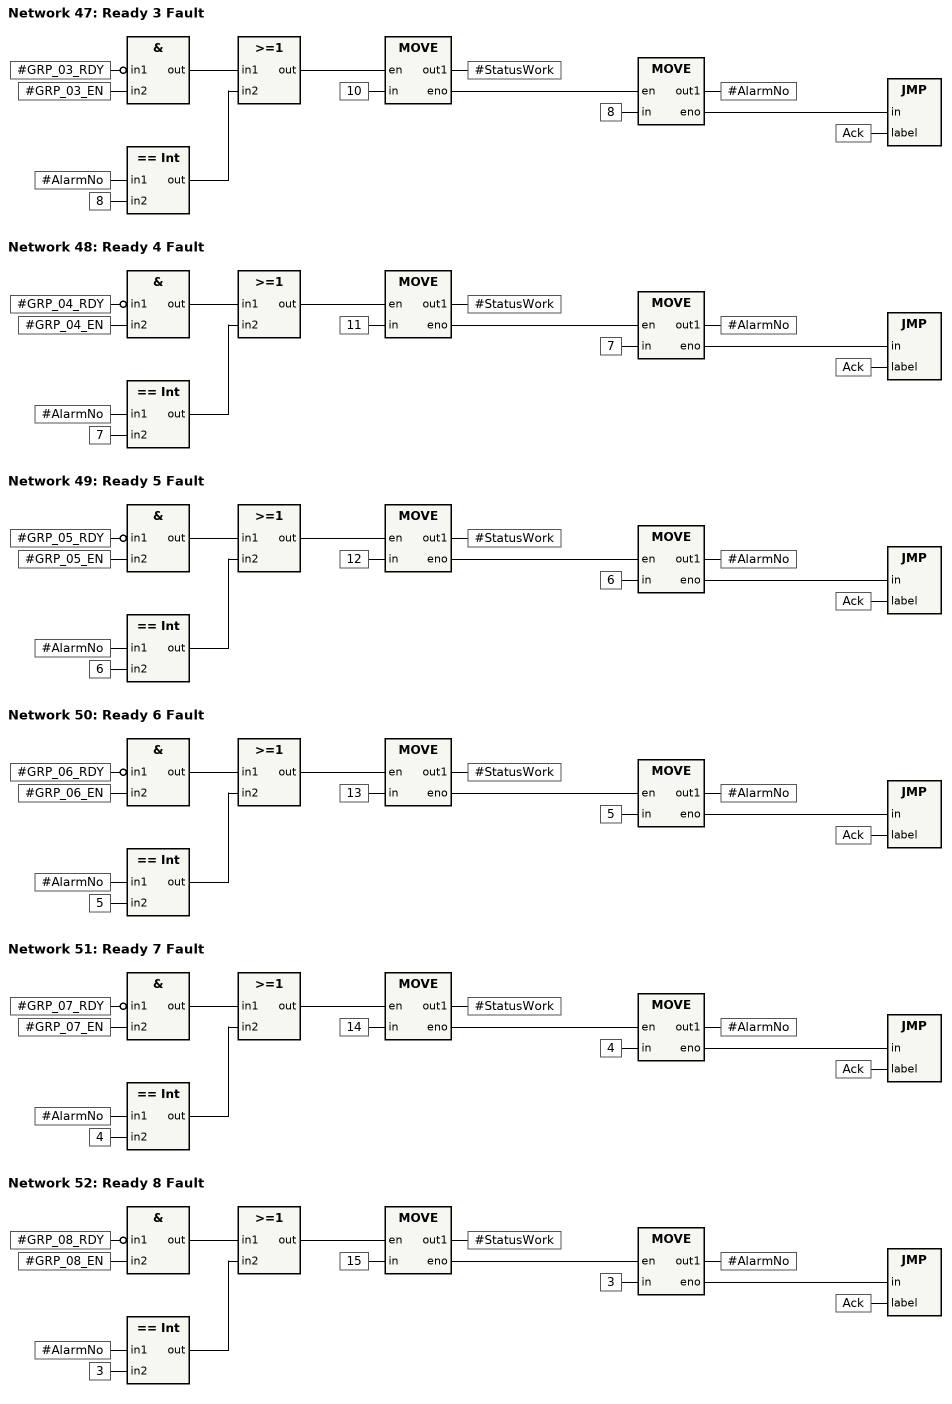
   // ENO of a box is taken as its EN; it also drops when the box reports an error
   #_w1 := (NOT #GRP_03_RDY AND #GRP_03_EN) OR (#AlarmNo = 8);
   IF #_w1 THEN
       #StatusWork := 10;
       #AlarmNo := 8;
       GOTO Ack;
   END_IF;
END_REGION

REGION Network 48: Ready 4 Fault
   // ENO of a box is taken as its EN; it also drops when the box reports an error
   #_w1 := (NOT #GRP_04_RDY AND #GRP_04_EN) OR (#AlarmNo = 7);
   IF #_w1 THEN
       #StatusWork := 11;
       #AlarmNo := 7;
       GOTO Ack;
   END_IF;
END_REGION

REGION Network 49: Ready 5 Fault
   // ENO of a box is taken as its EN; it also drops when the box reports an error
   #_w1 := (NOT #GRP_05_RDY AND #GRP_05_EN) OR (#AlarmNo = 6);
   IF #_w1 THEN
       #StatusWork := 12;
       #AlarmNo := 6;
       GOTO Ack;
   END_IF;
END_REGION

REGION Network 50: Ready 6 Fault
   // ENO of a box is taken as its EN; it also drops when the box reports an error
   #_w1 := (NOT #GRP_06_RDY AND #GRP_06_EN) OR (#AlarmNo = 5);
   IF #_w1 THEN
       #StatusWork := 13;
       #AlarmNo := 5;
       GOTO Ack;
   END_IF;
END_REGION

REGION Network 51: Ready 7 Fault
   // ENO of a box is taken as its EN; it also drops when the box reports an error
   #_w1 := (NOT #GRP_07_RDY AND #GRP_07_EN) OR (#AlarmNo = 4);
   IF #_w1 THEN
       #StatusWork := 14;
       #AlarmNo := 4;
       GOTO Ack;
   END_IF;
END_REGION

REGION Network 52: Ready 8 Fault
   // ENO of a box is taken as its EN; it also drops when the box reports an error
   #_w1 := (NOT #GRP_08_RDY AND #GRP_08_EN) OR (#AlarmNo = 3);
   IF #_w1 THEN
       #StatusWork := 15;
       #AlarmNo := 3;
       GOTO Ack;
   END_IF;
END_REGION

REGION Network 53: Ready 9 Fault
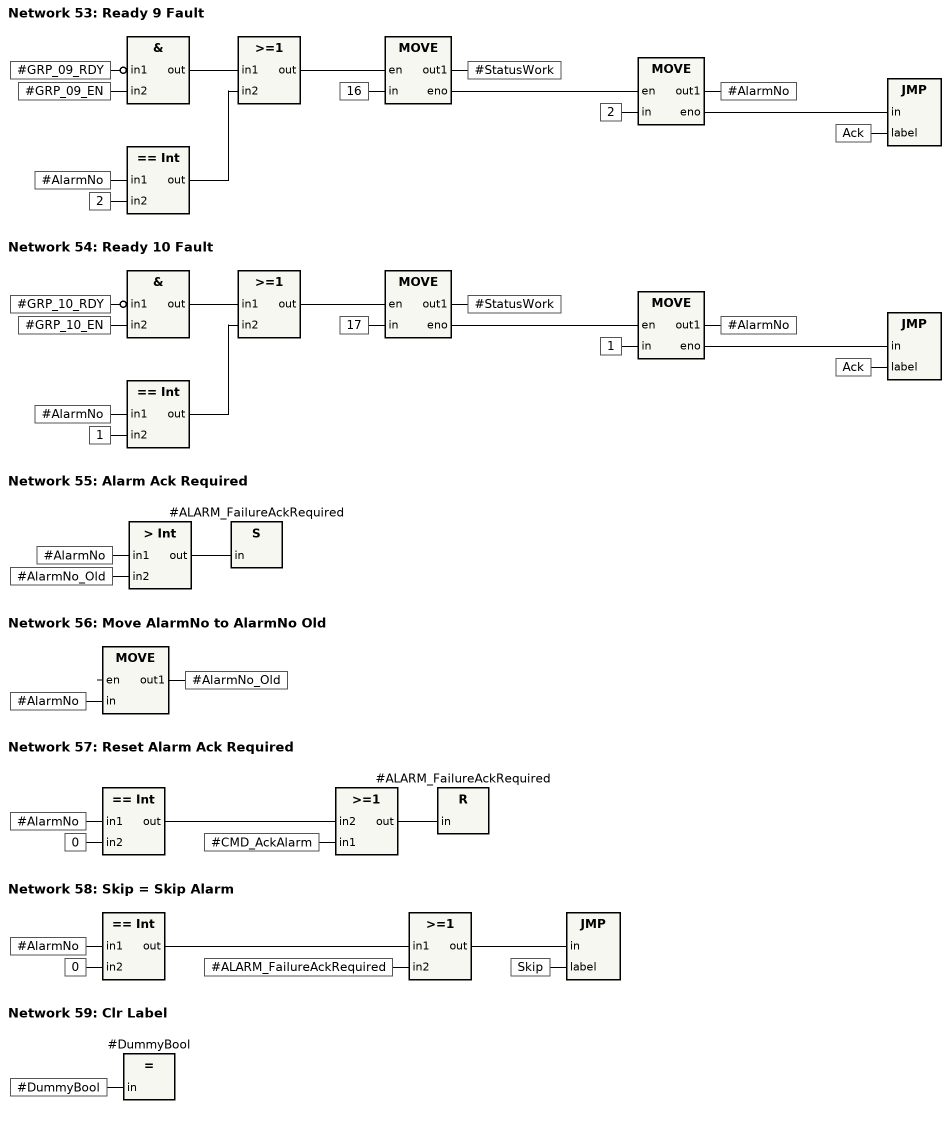
   // ENO of a box is taken as its EN; it also drops when the box reports an error
   #_w1 := (NOT #GRP_09_RDY AND #GRP_09_EN) OR (#AlarmNo = 2);
   IF #_w1 THEN
       #StatusWork := 16;
       #AlarmNo := 2;
       GOTO Ack;
   END_IF;
END_REGION

REGION Network 54: Ready 10 Fault
   // ENO of a box is taken as its EN; it also drops when the box reports an error
   #_w1 := (NOT #GRP_10_RDY AND #GRP_10_EN) OR (#AlarmNo = 1);
   IF #_w1 THEN
       #StatusWork := 17;
       #AlarmNo := 1;
       GOTO Ack;
   END_IF;
END_REGION

REGION Network 55: Alarm Ack Required
   Ack:
   IF #AlarmNo > #AlarmNo_Old THEN #ALARM_FailureAckRequired := TRUE; END_IF;
END_REGION

REGION Network 56: Move AlarmNo to AlarmNo Old
   #AlarmNo_Old := #AlarmNo;
END_REGION

REGION Network 57: Reset Alarm Ack Required
   IF (#AlarmNo = 0) OR #CMD_AckAlarm THEN #ALARM_FailureAckRequired := FALSE; END_IF;
END_REGION

REGION Network 58: Skip = Skip Alarm
   IF (#AlarmNo = 0) OR #ALARM_FailureAckRequired THEN GOTO Skip; END_IF;
END_REGION

REGION Network 59: Clr Label
   Clr:
   #DummyBool := #DummyBool;
END_REGION

REGION Network 60: Clear Alarm
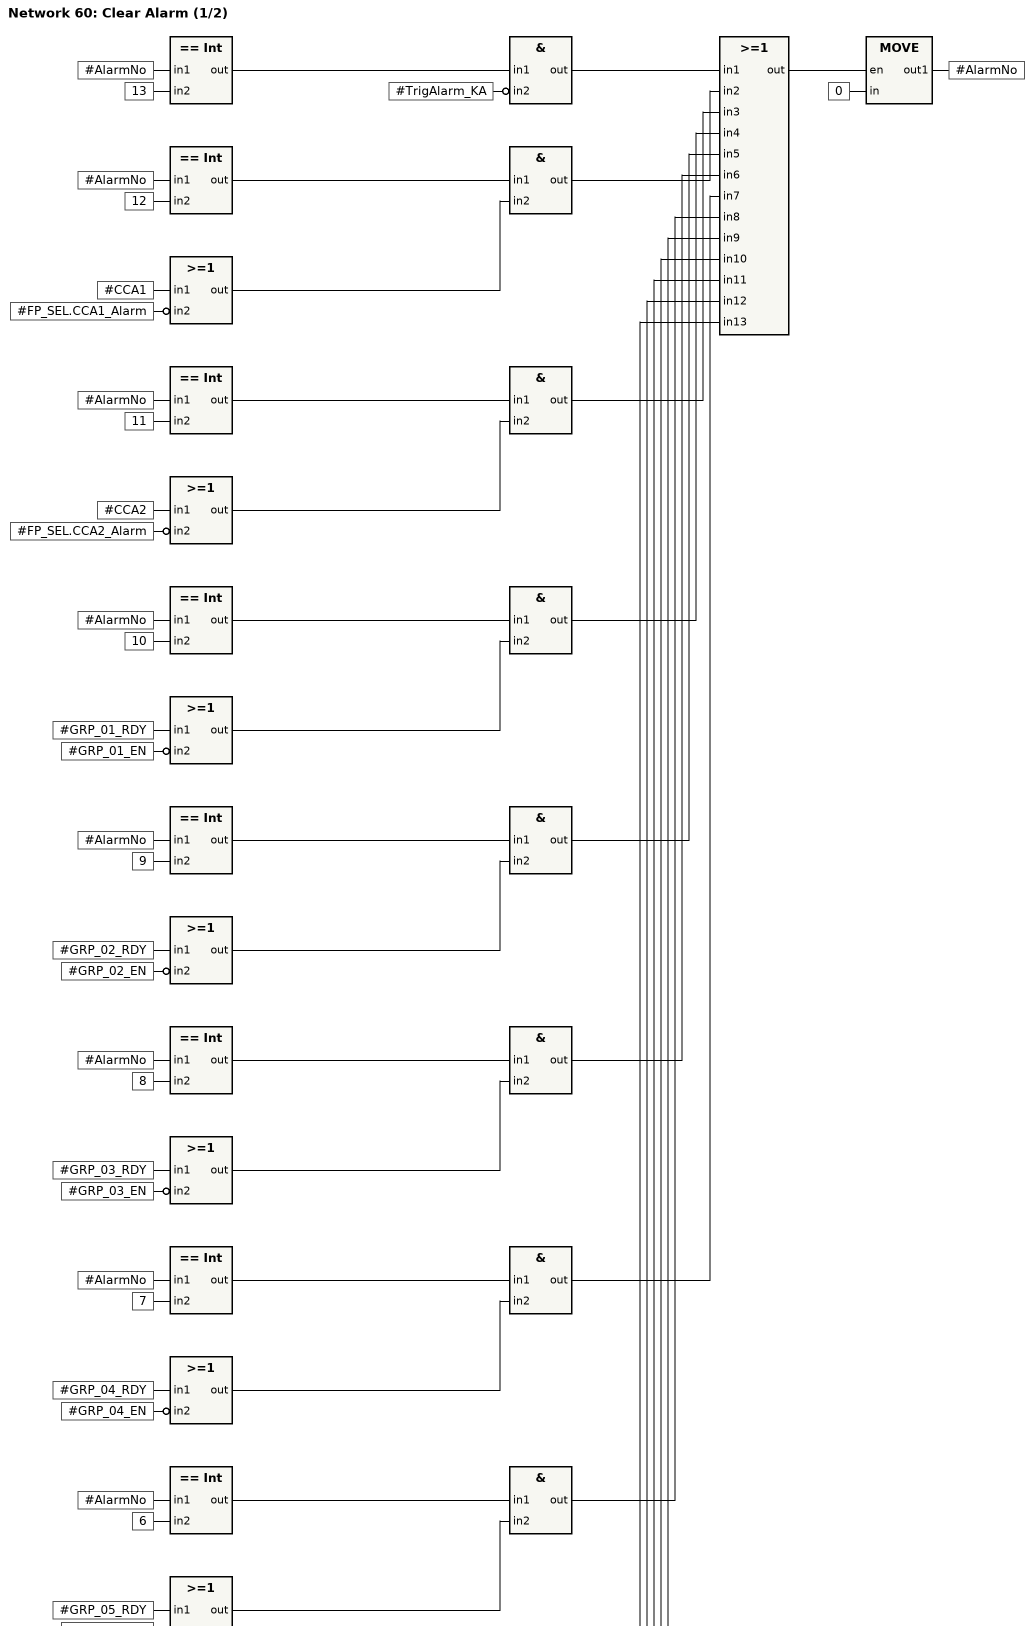
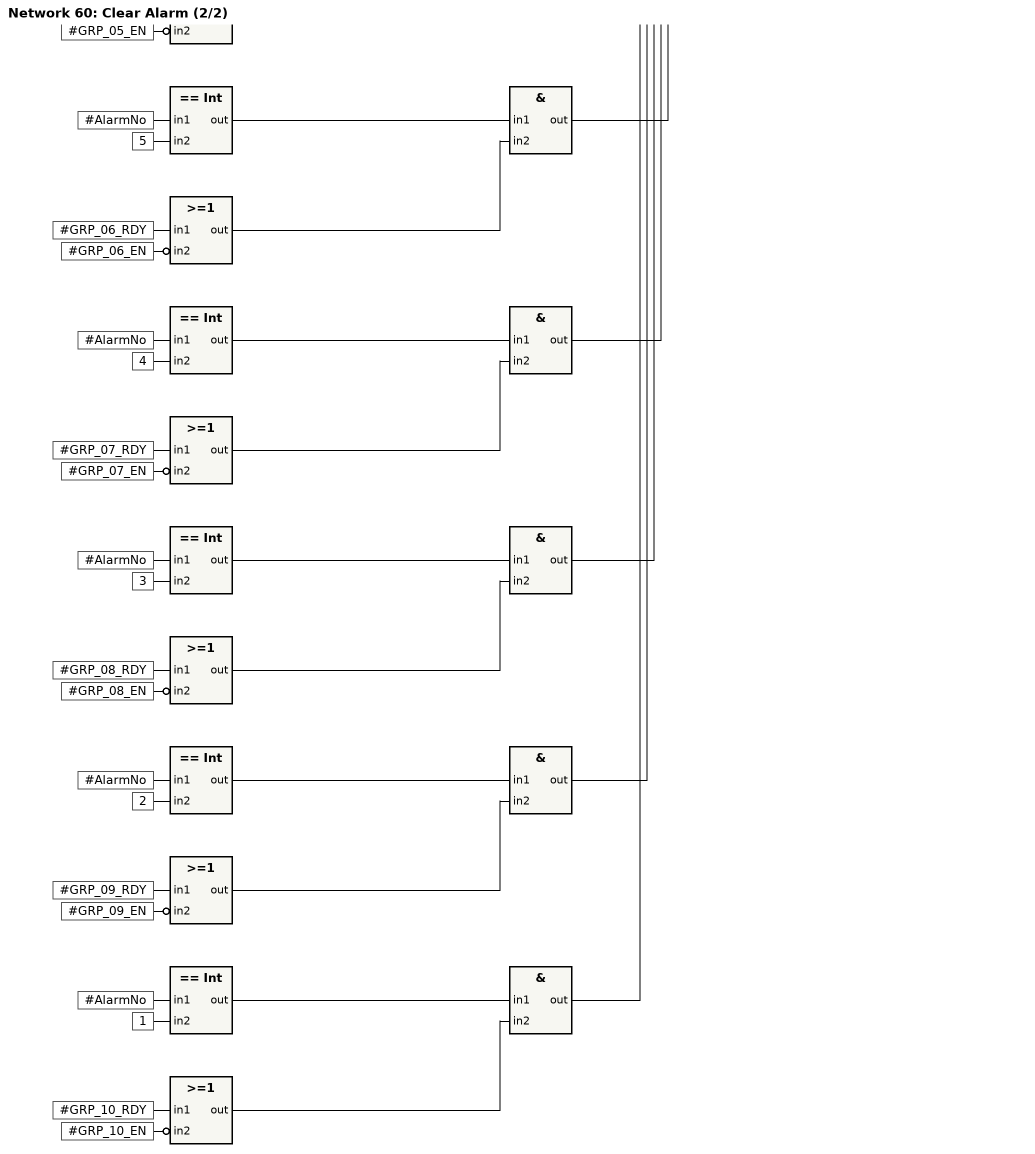
   IF ((#AlarmNo = 13) AND NOT #TrigAlarm_KA) OR ((#AlarmNo = 12) AND (#CCA1 OR NOT #FP_SEL.CCA1_Alarm)) OR ((#AlarmNo = 11) AND (#CCA2 OR NOT #FP_SEL.CCA2_Alarm)) OR ((#AlarmNo = 10) AND (#GRP_01_RDY OR NOT #GRP_01_EN)) OR ((#AlarmNo = 9) AND (#GRP_02_RDY OR NOT #GRP_02_EN)) OR ((#AlarmNo = 8) AND (#GRP_03_RDY OR NOT #GRP_03_EN)) OR ((#AlarmNo = 7) AND (#GRP_04_RDY OR NOT #GRP_04_EN)) OR ((#AlarmNo = 6) AND (#GRP_05_RDY OR NOT #GRP_05_EN)) OR ((#AlarmNo = 5) AND (#GRP_06_RDY OR NOT #GRP_06_EN)) OR ((#AlarmNo = 4) AND (#GRP_07_RDY OR NOT #GRP_07_EN)) OR ((#AlarmNo = 3) AND (#GRP_08_RDY OR NOT #GRP_08_EN)) OR ((#AlarmNo = 2) AND (#GRP_09_RDY OR NOT #GRP_09_EN)) OR ((#AlarmNo = 1) AND (#GRP_10_RDY OR NOT #GRP_10_EN)) THEN
       #AlarmNo := 0;
   END_IF;
END_REGION

REGION Network 61: Clear AlarmNo Old
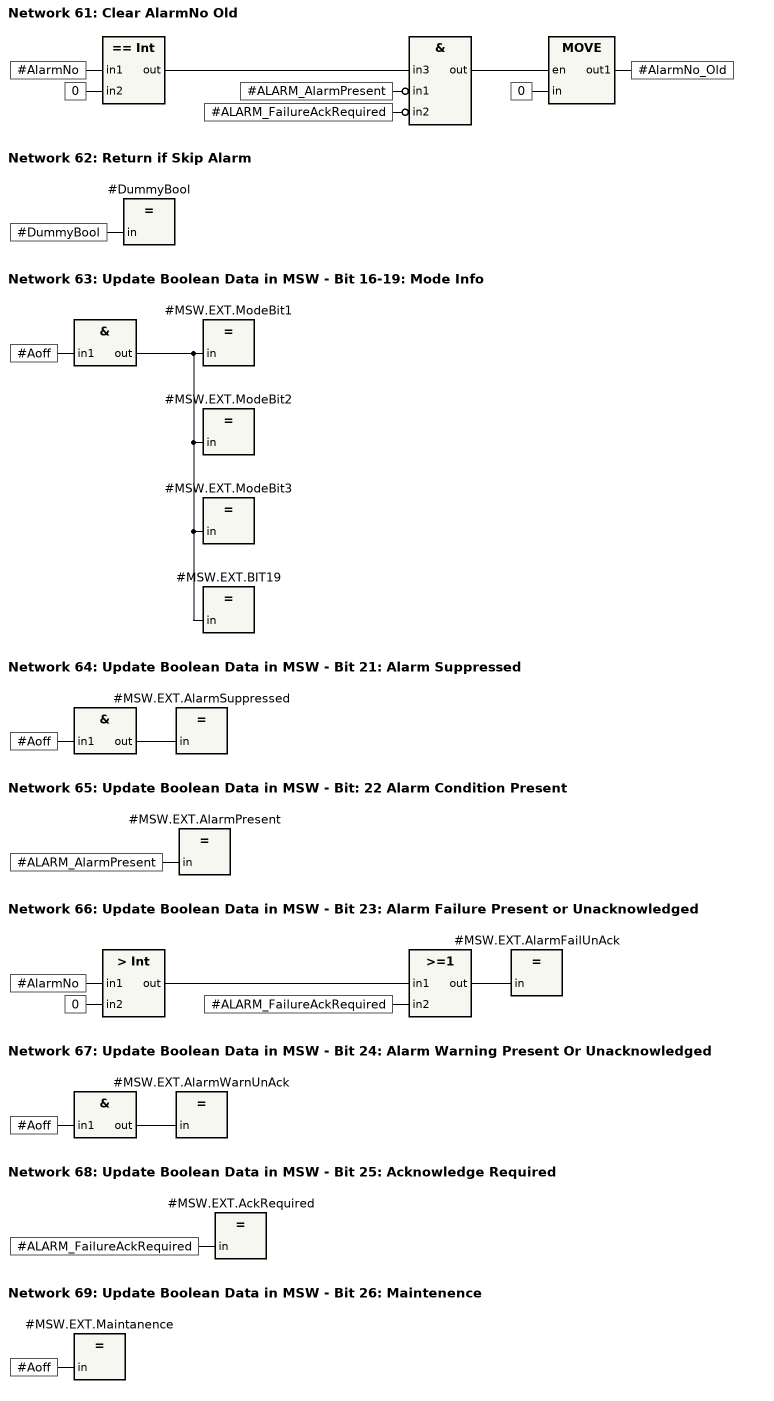
   IF (#AlarmNo = 0) AND NOT #ALARM_AlarmPresent AND NOT #ALARM_FailureAckRequired THEN
       #AlarmNo_Old := 0;
   END_IF;
END_REGION

REGION Network 62: Return if Skip Alarm
   Skip:
   #DummyBool := #DummyBool;
END_REGION

REGION Network 63: Update Boolean Data in MSW - Bit 16-19: Mode Info
   // 0 = Auto
   // 1= Single Start
   // 2 = Manual
   // 3= Local
   // 4= Test Mode
   #MSW.EXT.ModeBit1 := #Aoff;
   #MSW.EXT.ModeBit2 := #Aoff;
   #MSW.EXT.ModeBit3 := #Aoff;
   #MSW.EXT.BIT19 := #Aoff;
END_REGION

REGION Network 64: Update Boolean Data in MSW - Bit 21: Alarm Suppressed
   #MSW.EXT.AlarmSuppressed := #Aoff;
END_REGION

REGION Network 65: Update Boolean Data in MSW - Bit: 22 Alarm Condition Present
   #MSW.EXT.AlarmPresent := #ALARM_AlarmPresent;
END_REGION

REGION Network 66: Update Boolean Data in MSW - Bit 23: Alarm Failure Present or Unacknowledged
   #MSW.EXT.AlarmFailUnAck := (#AlarmNo > 0) OR #ALARM_FailureAckRequired;
END_REGION

REGION Network 67: Update Boolean Data in MSW - Bit 24: Alarm Warning Present Or Unacknowledged
   #MSW.EXT.AlarmWarnUnAck := #Aoff;
END_REGION

REGION Network 68: Update Boolean Data in MSW - Bit 25: Acknowledge Required
   #MSW.EXT.AckRequired := #ALARM_FailureAckRequired;
END_REGION

REGION Network 69: Update Boolean Data in MSW - Bit 26: Maintenence
   #MSW.EXT.Maintanence := #Aoff;
END_REGION

REGION Network 70: Update Boolean Data in MSW - Bit 27: Operation
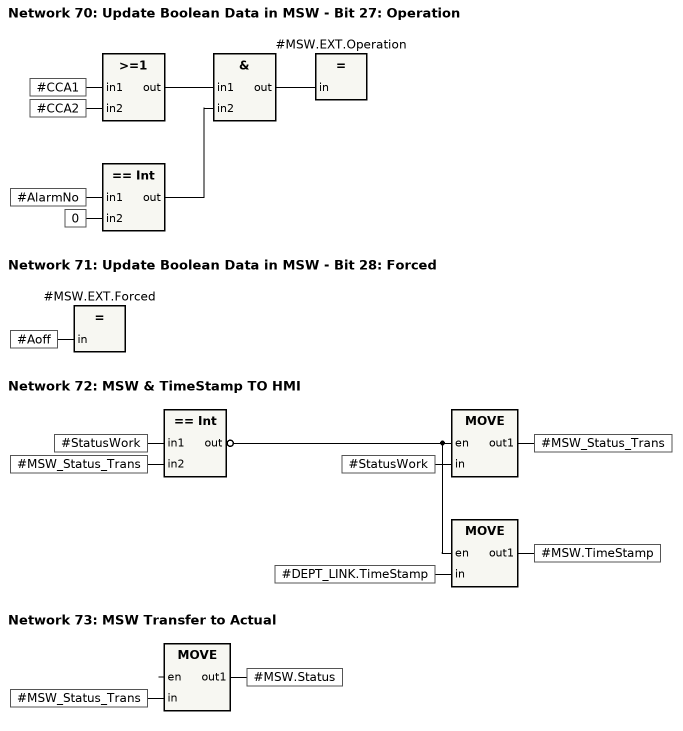
   #MSW.EXT.Operation := (#CCA1 OR #CCA2) AND (#AlarmNo = 0);
END_REGION

REGION Network 71: Update Boolean Data in MSW - Bit 28: Forced
   #MSW.EXT.Forced := #Aoff;
END_REGION

REGION Network 72: MSW & TimeStamp TO HMI
   #_w1 := NOT (#StatusWork = #MSW_Status_Trans);
   IF #_w1 THEN
       #MSW_Status_Trans := #StatusWork;
       #MSW.TimeStamp := #DEPT_LINK.TimeStamp;
   END_IF;
END_REGION

REGION Network 73: MSW Transfer to Actual
   #MSW.Status := #MSW_Status_Trans;
END_REGION
END_FUNCTION_BLOCK

FUNCTION_BLOCK "ACESYS_PLC_DIAG"   // FB222, FBD
TITLE = ACESYS V8.0 - Build 001 - PLC HW Diagnostic
{ S7_Optimized_Access := 'FALSE' }
AUTHOR : FLSmidth
FAMILY : ACESYS
NAME : PLC_DIAG
VERSION : 8.0
// Diagnostic of CPU Led status
// 
// ***SUPPORTED TYPES*** (Value of input parameter)
// Type "1500" and "1200"
// S7 - 151x/121x
// 
// *Diagnostic status*
// -RUN/STOP
// -ERROR
// -MAINT
   VAR_INPUT
      Master_Link : "ACESYS_MASTER_LINK";
      CPU_Type : Int;   // Valid NO: "1200", "1500"
   END_VAR
   VAR_OUTPUT
      CPU_OK : Bool;   // CPU Status OK
      Type_Fault : Bool;   // CPU Type Fault
      MSW : "ACESYS_HMI_STAT_32T";
   END_VAR
   VAR
      BlockInfo : Struct
         Ace_Version : Int;   // Acesys Block Version Number
         Ace_BuildNo : Int;   // Acesys Block Build Number
         DB_Number : Int;   // Block Instance DB Number
      END_STRUCT;
      FP_CMD : Struct   // Faceplate Commands
         Spare_08 : Bool;   // Bit8
         Spare_09 : Bool;   // Bit9
         Spare_10 : Bool;   // Bit10
         Spare_11 : Bool;   // Bit11
         Spare_12 : Bool;   // Bit12
         Spare_13 : Bool;   // Bit13
         Spare_14 : Bool;   // Bit14
         AckAlarm : Bool;   // Alarm Acknowledge
         Spare_00 : Bool;   // Bit0
         Spare_01 : Bool;   // Bit1
         Spare_02 : Bool;   // Bit2
         Spare_03 : Bool;   // Bit3
         Spare_04 : Bool;   // Bit4
         Spare_05 : Bool;   // Bit5
         Spare_06 : Bool;   // Bit6
         Spare_07 : Bool;   // Bit7
      END_STRUCT;
      FP_SHOW : Struct
         CPU_RUN_IND : Bool;
         Spare13 : Bool;
         Spare12 : Bool;
         Spare11 : Bool;
         Spare10 : Bool;
         Spare9 : Bool;
         Spare8 : Bool;
         Spare7 : Bool;
         Spare6 : Bool;
         Spare5 : Bool;
         Spare4 : Bool;
         CPU_MAINT : Bool;
         CPU_ERROR : Bool;
         Spare3 : Bool;
         Spare2 : Bool;
         Spare1 : Bool;
      END_STRUCT;
      StatusWork : Int;
      StatusBuilder : Int;
      SFC51_RET_VAL_Spare : Int;
      SFC51_BUSY_Spare : Bool;
      SZL_HEADER_Spare : Struct
         LENGTHDR : Word;
         N_DR : Word;
      END_STRUCT;
      Spare_W8 : Word;   // LED RUN Check
      Spare_W9 : Word;   // LED ERROR Check
      Spare_W10 : Word;   // LED MAINT Check
      Spare_W11 : Word;
      Spare_W12 : Word;
      Spare_W13 : Word;
      Spare_W14 : Word;
      Spare_W15 : Word;
      Record_LED_MAINT : Word;
      Spare_W16 : Word;
      Record_LED_ERROR : Word;
      Spare_W2 : Word;
      Spare_W3 : Word;
      Spare_W4 : Word;
      Spare_W5 : Word;
      Spare_W6 : Word;
      Spare_W7 : Word;
      AlarmNo : Int;
      AlarmNo_Old : Int;
      ALARM_AlarmPresent : Bool;
      ALARM_Failure_Ack_Requ : Bool;
      CMD_Acknowledge : Bool;   // Internal Acknowledge
      ALARM_SuppresionActiv : Bool;
      Type_1200 : Bool;   // Type 300 Selected
      Type_1500 : Bool;   // Type 400 Selected
      CPU_RUN_IND : Bool;   // CPU RUN Indicator Flashing=Run, Steady=Stopped/Error
      Spare25 : Bool;   // "1" = CPU LED OK
      Spare24 : Bool;   // "1" = CPU LED OK
      Spare23 : Bool;
      Spare22 : Bool;
      Spare21 : Bool;
      Spare20 : Bool;
      Spare19 : Bool;
      Spare18 : Bool;
      CPU_MAINT : Bool;
      Spare16 : Bool;
      CPU_ERROR : Bool;
      Spare14 : Bool;
      Spare13 : Bool;
      Spare12 : Bool;
      Spare11 : Bool;
      Spare10 : Bool;
      Spare9 : Bool;
      Spare8 : Bool;
      Spare7 : Bool;
      Spare6 : Bool;
      Spare5 : Bool;
      Spare4 : Bool;
      Spare3 : Bool;
      Spare2 : Bool;
      Spare1 : Bool;
      OUT : Struct
         CPU_OK : Bool;
         Type_Fault : Bool;
      END_STRUCT;
      MSW_Status_Trans : Int;
   END_VAR
   VAR_TEMP
      LED_Record_Word1 : Word;   // LED Record
      LED_Record_Word2 : Word;   // LED Record
      LED_Record_Word3 : Word;   // LED Record
      LED_Record_Word4 : Word;   // LED Record
      LED_Record_Word5 : Word;   // LED Record
      LED_Record_Word6 : Word;   // LED Record
      LED_Record_Word7 : Word;   // LED Record
      LED_Record_Word8 : Word;   // LED Record
      LED_Record_Word9 : Word;   // LED Record
      LED_Record_Word10 : Word;   // LED Record
      AOn : Bool;   // Always On
      AOff : Bool;   // Always Off
      dummybool : Bool;
      Status_Add : Int;
   END_VAR
   VAR_TEMP   // added for the SCL form of the ladder/FBD networks
      _w1 : Bool;
   END_VAR
BEGIN

REGION Network 1: Always On
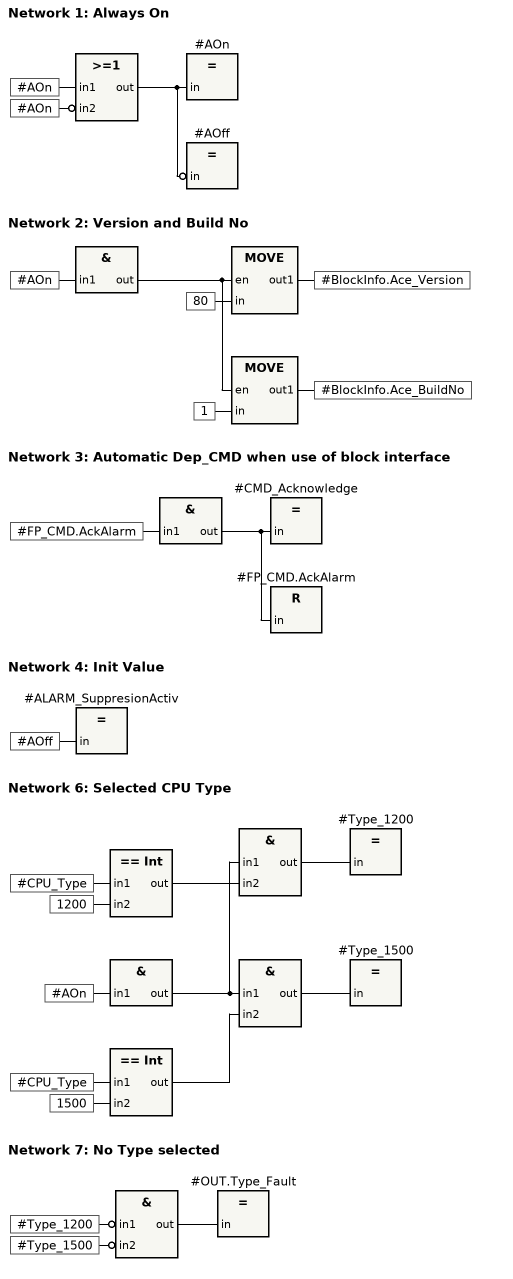
   #AOn := #AOn OR NOT #AOn;
   #AOff := NOT #AOn;
END_REGION

REGION Network 2: Version and Build No
   IF #AOn THEN
       #BlockInfo.Ace_Version := 80;
       #BlockInfo.Ace_BuildNo := 1;
   END_IF;
END_REGION

REGION Network 3: Automatic Dep_CMD when use of block interface
   #CMD_Acknowledge := #FP_CMD.AckAlarm;
   IF #FP_CMD.AckAlarm THEN #FP_CMD.AckAlarm := FALSE; END_IF;
END_REGION

REGION Network 4: Init Value
   #ALARM_SuppresionActiv := #AOff;
END_REGION

REGION Network 5 (STL): Instance DB Number to Faceplate
         L     DINO;
         T     #BlockInfo.DB_Number;
END_REGION

REGION Network 6: Selected CPU Type
   #Type_1200 := #AOn AND (#CPU_Type = 1200);
   #Type_1500 := #AOn AND (#CPU_Type = 1500);
END_REGION

REGION Network 7: No Type selected
   #OUT.Type_Fault := NOT #Type_1200 AND NOT #Type_1500;
END_REGION

REGION Network 8: Set Show Parameter
   // - From 300/400 Series LED status, not available or not used LED's are given '0' for 1200/1500
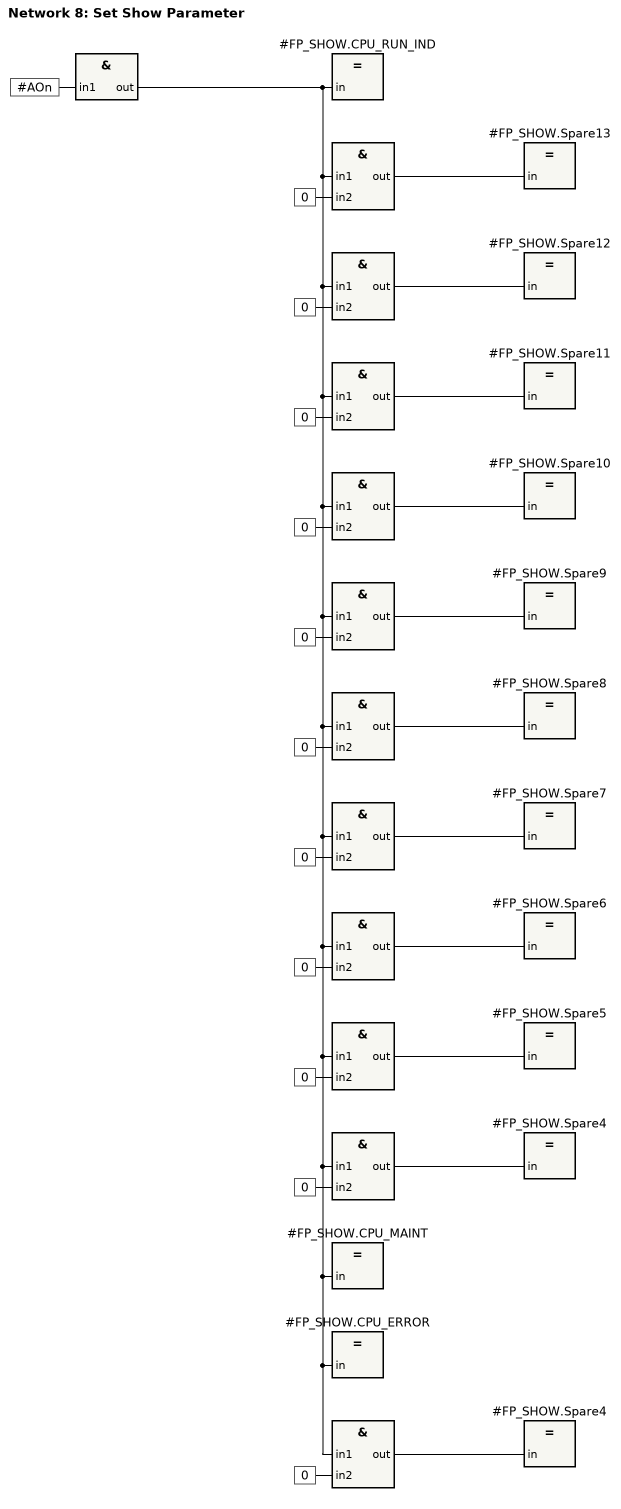
   #FP_SHOW.CPU_RUN_IND := #AOn;
   #FP_SHOW.Spare13 := #AOn AND 0;
   #FP_SHOW.Spare12 := #AOn AND 0;
   #FP_SHOW.Spare11 := #AOn AND 0;
   #FP_SHOW.Spare10 := #AOn AND 0;
   #FP_SHOW.Spare9 := #AOn AND 0;
   #FP_SHOW.Spare8 := #AOn AND 0;
   #FP_SHOW.Spare7 := #AOn AND 0;
   #FP_SHOW.Spare6 := #AOn AND 0;
   #FP_SHOW.Spare5 := #AOn AND 0;
   #FP_SHOW.Spare4 := #AOn AND 0;
   #FP_SHOW.CPU_MAINT := #AOn;
   #FP_SHOW.CPU_ERROR := #AOn;
   #FP_SHOW.Spare4 := #AOn AND 0;
END_REGION

REGION Network 9: CPU_ERROR LED Indication
   // 0 = LED does not exist or status information not available
   // 1 = Permanently switched off
   // 2 = Color 1 (e.g., for LED STOP/RUN: green) permanently ON
   // 3 = Color 2 (e.g., for LED STOP/RUN: orange) permanently ON
   // 4 = Color 1 flashing at 2 Hz
   // 5 = Color 2 flashing at 2 Hz
   // 6 = Colors 1 and 2 flashing alternately at 2 Hz
   // 7 = LED is active, color 1
   // 8 = LED is active, color 2
   // 9 = LED does not exist or status information not available
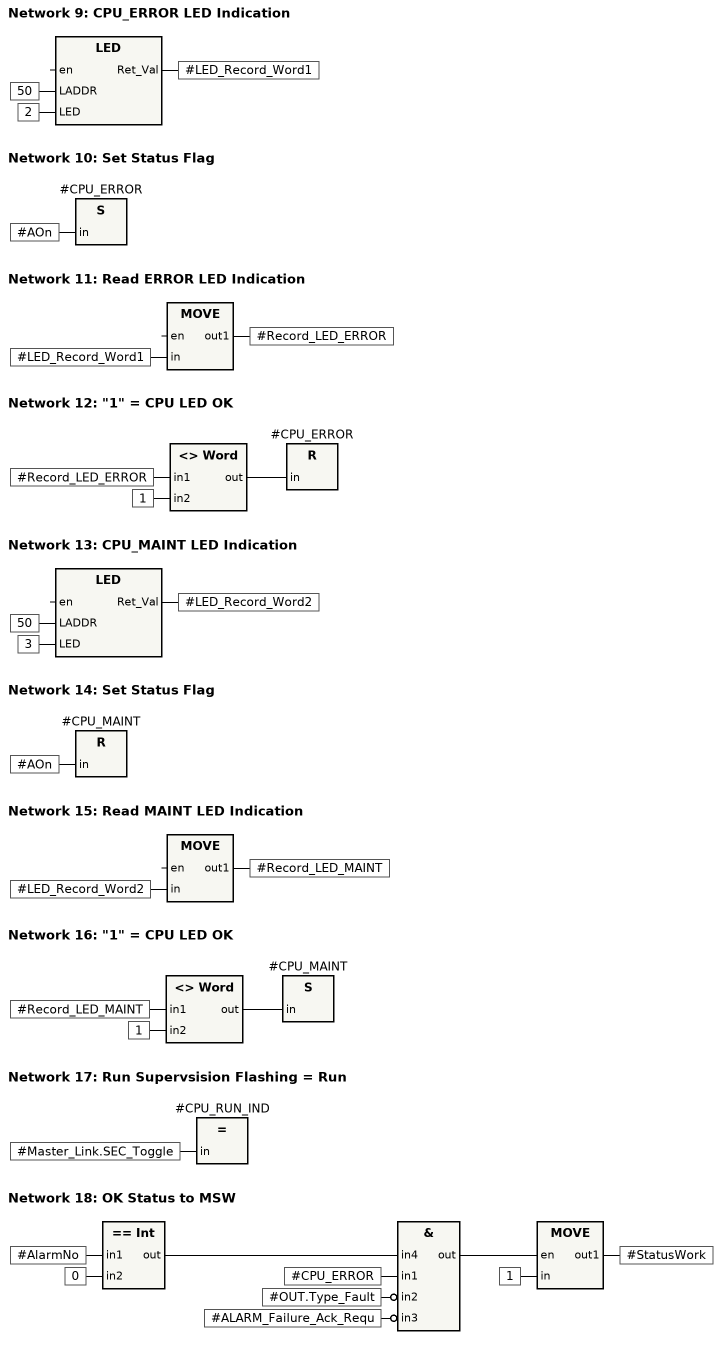
   #LED_Record_Word1 := LED(LADDR := 50, LED := 2);
END_REGION

REGION Network 10: Set Status Flag
   IF #AOn THEN #CPU_ERROR := TRUE; END_IF;
END_REGION

REGION Network 11: Read ERROR LED Indication
   #Record_LED_ERROR := #LED_Record_Word1;
END_REGION

REGION Network 12: "1" = CPU LED OK
   IF #Record_LED_ERROR <> 1 THEN #CPU_ERROR := FALSE; END_IF;
END_REGION

REGION Network 13: CPU_MAINT LED Indication
   // This LED indicates Maintenance required OR Force Job Active
   #LED_Record_Word2 := LED(LADDR := 50, LED := 3);
END_REGION

REGION Network 14: Set Status Flag
   IF #AOn THEN #CPU_MAINT := FALSE; END_IF;
END_REGION

REGION Network 15: Read MAINT LED Indication
   #Record_LED_MAINT := #LED_Record_Word2;
END_REGION

REGION Network 16: "1" = CPU LED OK
   IF #Record_LED_MAINT <> 1 THEN #CPU_MAINT := TRUE; END_IF;
END_REGION

REGION Network 17: Run Supervsision Flashing = Run
   #CPU_RUN_IND := #Master_Link.SEC_Toggle;
END_REGION

REGION Network 18: OK Status to MSW
   IF (#AlarmNo = 0) AND #CPU_ERROR AND NOT #OUT.Type_Fault AND NOT #ALARM_Failure_Ack_Requ THEN
       #StatusWork := 1;
   END_IF;
END_REGION

REGION Network 19: Skip alarm handling if Emergency Stop or no alarm present
   // Skip = Skip Alarm
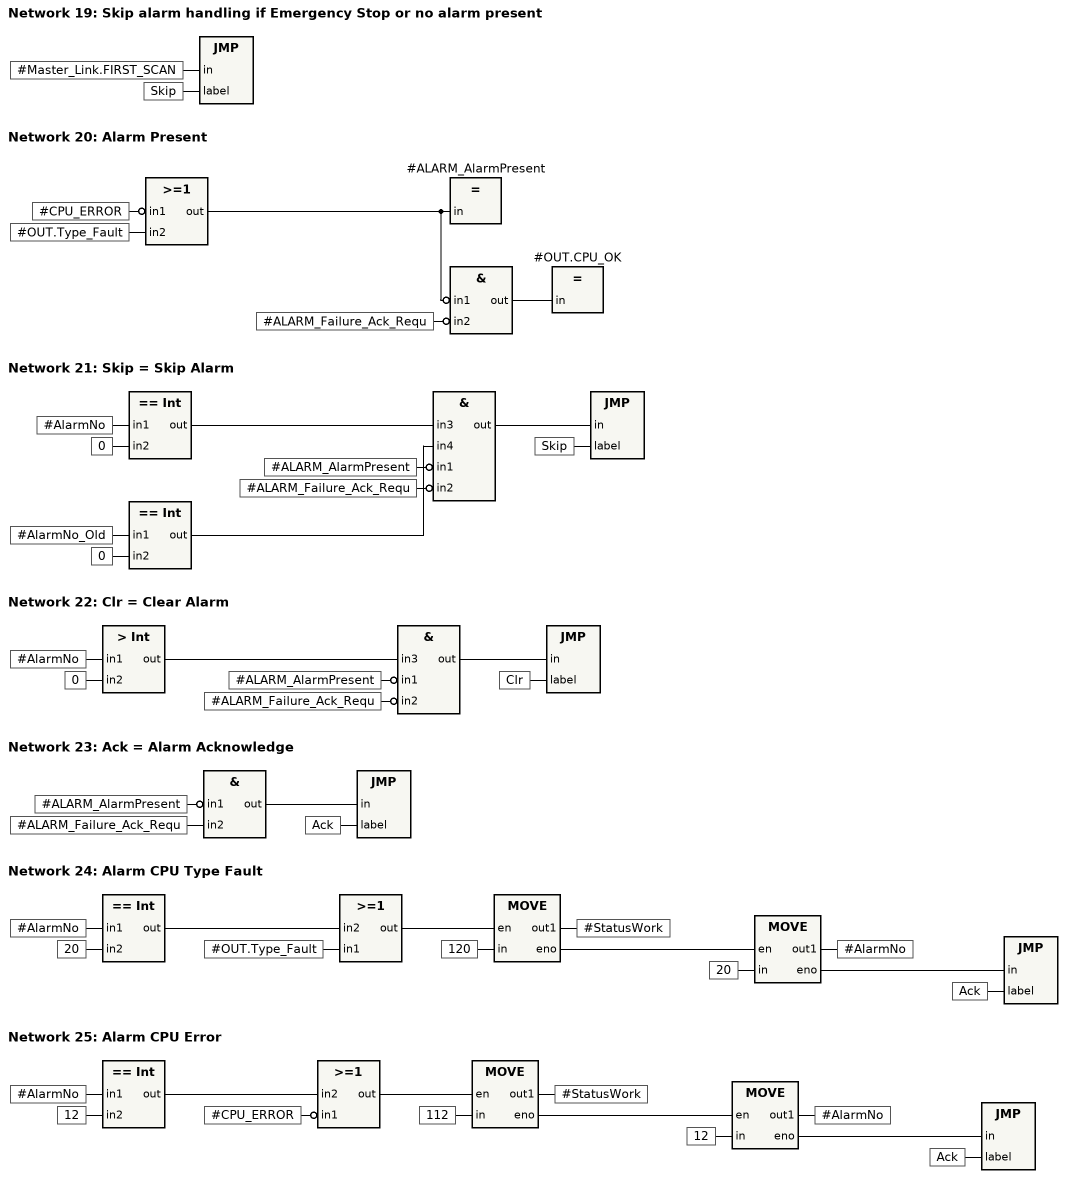
   IF #Master_Link.FIRST_SCAN THEN GOTO Skip; END_IF;
END_REGION

REGION Network 20: Alarm Present
   #ALARM_AlarmPresent := NOT #CPU_ERROR OR #OUT.Type_Fault;
   #OUT.CPU_OK := NOT #ALARM_AlarmPresent AND NOT #ALARM_Failure_Ack_Requ;
END_REGION

REGION Network 21: Skip = Skip Alarm
   IF (#AlarmNo = 0) AND (#AlarmNo_Old = 0) AND NOT #ALARM_AlarmPresent AND NOT #ALARM_Failure_Ack_Requ THEN
       GOTO Skip;
   END_IF;
END_REGION

REGION Network 22: Clr = Clear Alarm
   IF (#AlarmNo > 0) AND NOT #ALARM_AlarmPresent AND NOT #ALARM_Failure_Ack_Requ THEN GOTO Clr; END_IF;
END_REGION

REGION Network 23: Ack = Alarm Acknowledge
   IF NOT #ALARM_AlarmPresent AND #ALARM_Failure_Ack_Requ THEN GOTO Ack; END_IF;
END_REGION

REGION Network 24: Alarm CPU Type Fault
   // ENO of a box is taken as its EN; it also drops when the box reports an error
   #_w1 := (#AlarmNo = 20) OR #OUT.Type_Fault;
   IF #_w1 THEN
       #StatusWork := 120;
       #AlarmNo := 20;
       GOTO Ack;
   END_IF;
END_REGION

REGION Network 25: Alarm CPU Error
   // ENO of a box is taken as its EN; it also drops when the box reports an error
   #_w1 := (#AlarmNo = 12) OR NOT #CPU_ERROR;
   IF #_w1 THEN
       #StatusWork := 112;
       #AlarmNo := 12;
       GOTO Ack;
   END_IF;
END_REGION

REGION Network 26: Alarm Acknowledge
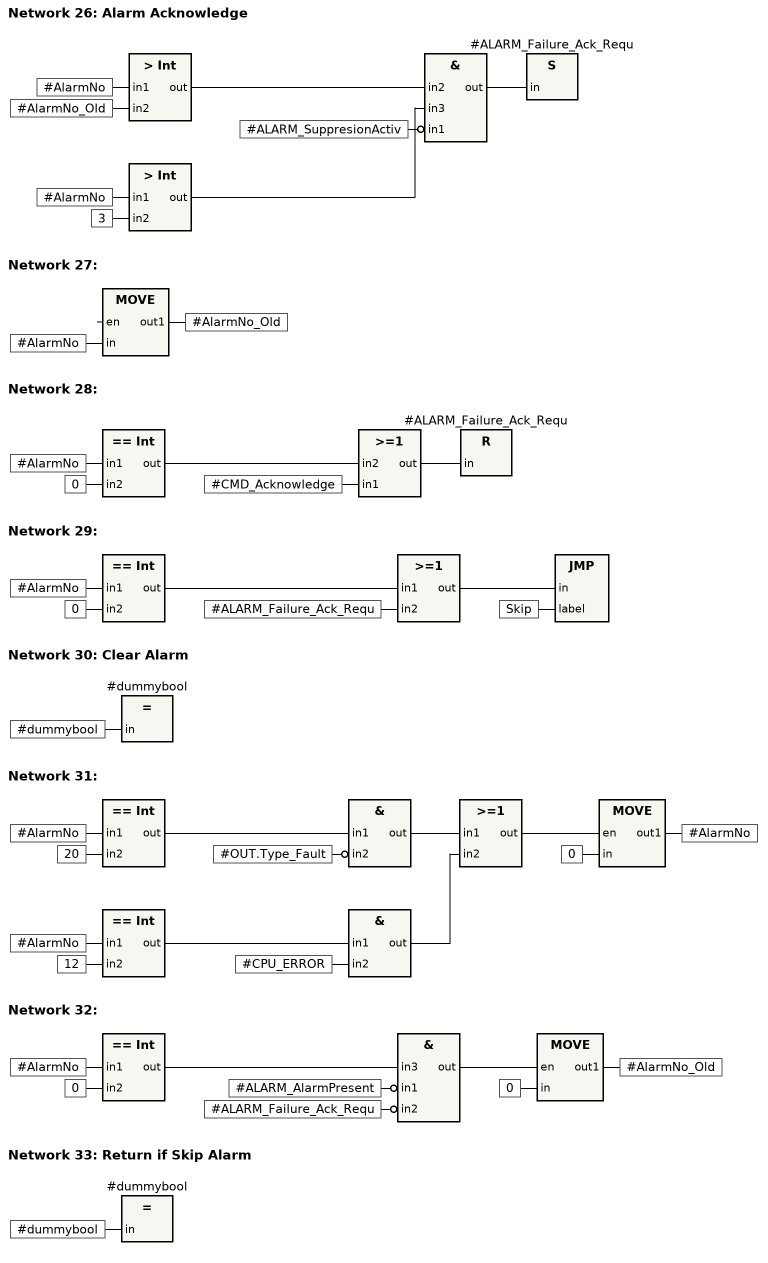
   Ack:
   IF (#AlarmNo > #AlarmNo_Old) AND (#AlarmNo > 3) AND NOT #ALARM_SuppresionActiv THEN
       #ALARM_Failure_Ack_Requ := TRUE;
   END_IF;
END_REGION

REGION Network 27
   #AlarmNo_Old := #AlarmNo;
END_REGION

REGION Network 28
   IF (#AlarmNo = 0) OR #CMD_Acknowledge THEN #ALARM_Failure_Ack_Requ := FALSE; END_IF;
END_REGION

REGION Network 29
   // Skip = Skip Alarm
   IF (#AlarmNo = 0) OR #ALARM_Failure_Ack_Requ THEN GOTO Skip; END_IF;
END_REGION

REGION Network 30: Clear Alarm
   Clr:
   #dummybool := #dummybool;
END_REGION

REGION Network 31
   IF ((#AlarmNo = 20) AND NOT #OUT.Type_Fault) OR ((#AlarmNo = 12) AND #CPU_ERROR) THEN
       #AlarmNo := 0;
   END_IF;
END_REGION

REGION Network 32
   IF (#AlarmNo = 0) AND NOT #ALARM_AlarmPresent AND NOT #ALARM_Failure_Ack_Requ THEN
       #AlarmNo_Old := 0;
   END_IF;
END_REGION

REGION Network 33: Return if Skip Alarm
   Skip:
   #dummybool := #dummybool;
END_REGION

REGION Network 34: Bit 16-19: Mode
   // 0 = Auto
   // 1= Single Start
   // 2 = Manual
   // 3= Local
   // 4= Test Mode
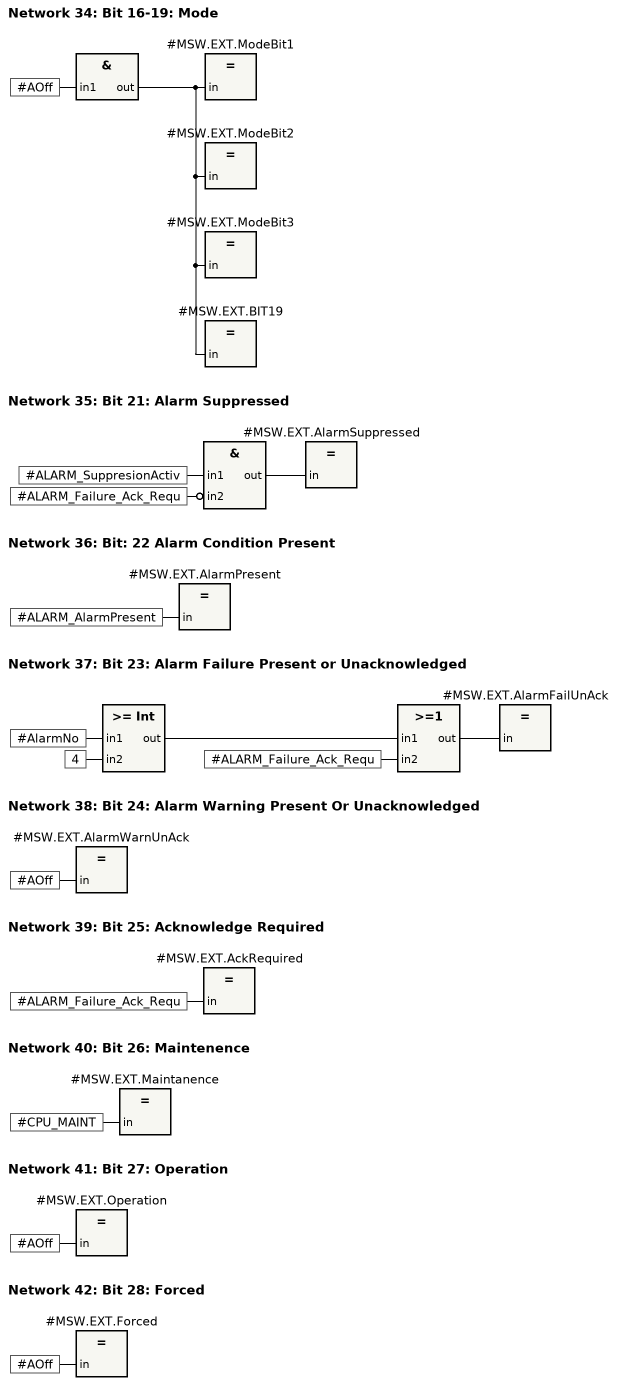
   #MSW.EXT.ModeBit1 := #AOff;
   #MSW.EXT.ModeBit2 := #AOff;
   #MSW.EXT.ModeBit3 := #AOff;
   #MSW.EXT.BIT19 := #AOff;
END_REGION

REGION Network 35: Bit 21: Alarm Suppressed
   #MSW.EXT.AlarmSuppressed := #ALARM_SuppresionActiv AND NOT #ALARM_Failure_Ack_Requ;
END_REGION

REGION Network 36: Bit: 22 Alarm Condition Present
   #MSW.EXT.AlarmPresent := #ALARM_AlarmPresent;
END_REGION

REGION Network 37: Bit 23: Alarm Failure Present or Unacknowledged
   #MSW.EXT.AlarmFailUnAck := (#AlarmNo >= 4) OR #ALARM_Failure_Ack_Requ;
END_REGION

REGION Network 38: Bit 24: Alarm Warning Present Or Unacknowledged
   #MSW.EXT.AlarmWarnUnAck := #AOff;
END_REGION

REGION Network 39: Bit 25: Acknowledge Required
   #MSW.EXT.AckRequired := #ALARM_Failure_Ack_Requ;
END_REGION

REGION Network 40: Bit 26: Maintenence
   #MSW.EXT.Maintanence := #CPU_MAINT;
END_REGION

REGION Network 41: Bit 27: Operation
   #MSW.EXT.Operation := #AOff;
END_REGION

REGION Network 42: Bit 28: Forced
   #MSW.EXT.Forced := #AOff;
END_REGION

REGION Network 43
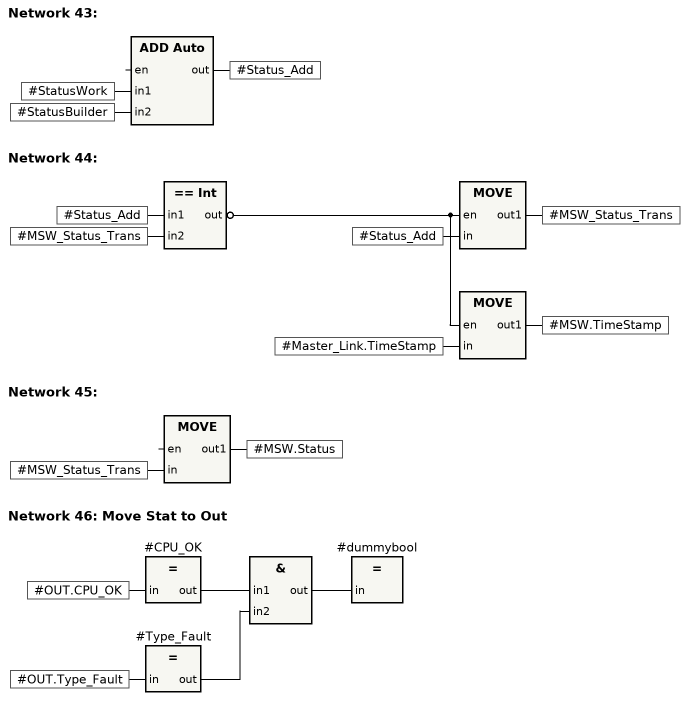
   #Status_Add := #StatusWork + #StatusBuilder;
END_REGION

REGION Network 44
   #_w1 := NOT (#Status_Add = #MSW_Status_Trans);
   IF #_w1 THEN
       #MSW_Status_Trans := #Status_Add;
       #MSW.TimeStamp := #Master_Link.TimeStamp;
   END_IF;
END_REGION

REGION Network 45
   #MSW.Status := #MSW_Status_Trans;
END_REGION

REGION Network 46: Move Stat to Out
   #CPU_OK := #OUT.CPU_OK;
   #Type_Fault := #OUT.Type_Fault;
   #dummybool := #OUT.CPU_OK AND #OUT.Type_Fault;
END_REGION
END_FUNCTION_BLOCK

FUNCTION_BLOCK "ACESYS_PROFINET"   // FB223, FBD
TITLE = ACESYS V8.0 - Build 001 - Profinet Diagnostic
{ S7_Optimized_Access := 'FALSE' }
VERSION : 0.1
// Diagnostic of ProfiNet nodes 1-256
// -Detect configured node (Configured in HW Config)
// -Detect Present Node (Node Present on Net)
// -Detect affected node with error (Node affected)
// 
// - Parameter: IO_System_CP refering to HW configuration
// - Internal Alarm handling for nodes
// 
// Bit [0] in array:
// CONFIGURED
// PRESENT
// AFFECTED
// is sum bit for all nodes in struct
   VAR_INPUT
      Master_Link : "ACESYS_MASTER_LINK";
      IO_System_CP : Int;   // CP IO System number
   END_VAR
   VAR_OUTPUT
      MSW : "ACESYS_HMI_STAT_32T";
   END_VAR
   VAR
      BlockInfo : Struct   // Faceplate Block Info
         Ace_Version : Int;   // Acesys Block Version Number
         Ace_BuildNo : Int;   // Acesys Block Build Number
         DB_Number : Int;   // Block Instance DB Number
      END_STRUCT;
      FP_CMD : Struct   // Faceplate Commands
         Spare_08 : Bool;   // Bit8
         Spare_09 : Bool;   // Bit9
         Spare_10 : Bool;   // Bit10
         Spare_11 : Bool;   // Bit11
         Spare_12 : Bool;   // Bit12
         Spare_13 : Bool;   // Bit13
         Spare_14 : Bool;   // Bit14
         AckAlarm : Bool;   // Alarm Acknowledge
         Spare_00 : Bool;   // Bit0
         Spare_01 : Bool;   // Bit1
         Spare_02 : Bool;   // Bit2
         Spare_03 : Bool;   // Bit3
         Spare_04 : Bool;   // Bit4
         Spare_05 : Bool;   // Bit5
         Spare_06 : Bool;   // Bit6
         Spare_07 : Bool;   // Bit7
      END_STRUCT;
      FP_PARM : Struct   // Faceplate Parameters
         SLAVES_AFFECTED_NUM : Int;
         SLAVES_EXIST_NUM : Int;
      END_STRUCT;
      INDEX_CONFIG_Spare : Word;   // Spare
      CONFIGURED : Array[0..257] of Bool;   // Configured Nodes, 1 = Rack/Device Configured
      INDEX_PRESENT_Spare : Word;   // Spare
      PRESENT : Array[0..257] of Bool;   // Present Nodes, 1 = Rack/Device Present
      INDEX_AFFECTED_Spare : Word;   // Spare
      AFFECTED : Array[0..257] of Bool;   // Affected Nodes, 1 = failed
      READING_FAILURE : Bool;   // Wrong or unknown Mode OR no CPU Supported
      READING_INDEX_FAILURE : Bool;   // Wrong or non permited Hardware ID
      BUSY_READ_SZL_094_Spare : Bool;   // Spare
      BUSY_READ_SZL_294_Spare : Bool;   // Spare
      BUSY_READ_SZL_694_Spare : Bool;   // Spare
      DONE_READ_SZL_094_Spare : Bool;   // Spare
      DONE_READ_SZL_294_Spare : Bool;   // Spare
      DONE_READ_SZL_694_Spare : Bool;   // Spare
      DR_Data : Array[0..129] of Word;   // Device States Data
      DR_Data_Trans AT DR_Data : Array[0..2079] of Bool;
      ALARM_AlarmPresent : Bool;
      ALARM_Failure_Ack_Requ : Bool;
      ConfigNodeAlarm : Bool;   // No Node Configured on NW
      NodeErrorAlarm : Bool;   // Node Affected on NW
      ALARM_SuppresionActiv : Bool;
      CMD_Acknowledge : Bool;   // Internal Acknowledge
      Spare10 : Bool;
      Spare9 : Bool;
      Spare8 : Bool;
      Spare7 : Bool;
      Spare6 : Bool;
      Spare5 : Bool;
      Spare4 : Bool;
      Spare3 : Bool;
      Spare2 : Bool;
      Spare1 : Bool;
      AlarmNo : Int;
      AlarmNo_Old : Int;
      StatusWork : Int;
      MSW_Status_Trans : Int;
   END_VAR
   VAR_TEMP
      AOn : Bool;   // Always On
      AOff : Bool;   // Always Off
      OFFSET : Int;
      RETVAL_DEVICE : Int;
      slaves_affected_number : Int;
      slaves_Present_number : Int;
      dummybool : Bool;
      GeoAddr : GEOADDR;   // Structure for reading Hardware ID from PN Master No
      HW_ID : Hw_Any;
      RETVAL_GEO : Int;
      RETVAL_DEVICE_1 : Int;
      RETVAL_DEVICE_2 : Int;
   END_VAR
   VAR_TEMP   // added for the SCL form of the ladder/FBD networks
      _w1 : Bool;
   END_VAR
BEGIN

REGION Network 1: Always On
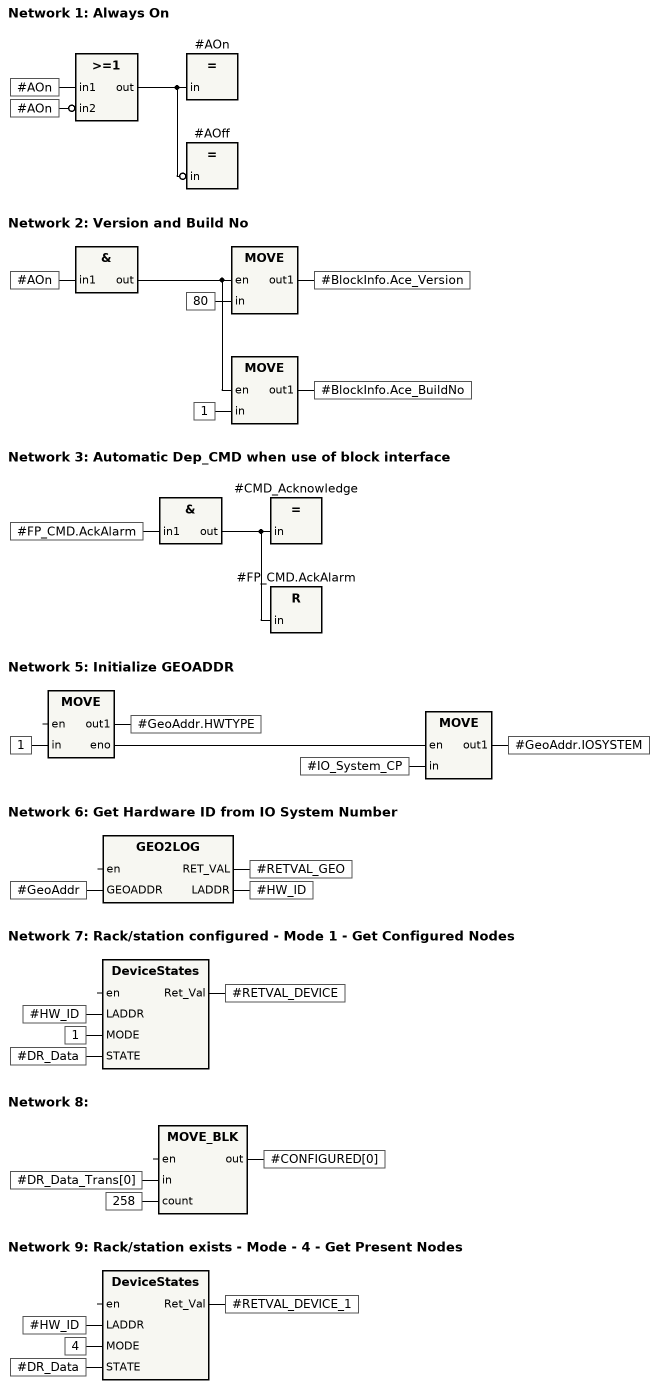
   #AOn := #AOn OR NOT #AOn;
   #AOff := NOT #AOn;
END_REGION

REGION Network 2: Version and Build No
   IF #AOn THEN
       #BlockInfo.Ace_Version := 80;
       #BlockInfo.Ace_BuildNo := 1;
   END_IF;
END_REGION

REGION Network 3: Automatic Dep_CMD when use of block interface
   #CMD_Acknowledge := #FP_CMD.AckAlarm;
   IF #FP_CMD.AckAlarm THEN #FP_CMD.AckAlarm := FALSE; END_IF;
END_REGION

REGION Network 4 (STL): Instance DB Number to Faceplate
         L     DINO;
         T     #BlockInfo.DB_Number;
END_REGION

REGION Network 5: Initialize GEOADDR
   // ENO of a box is taken as its EN; it also drops when the box reports an error
   #GeoAddr.HWTYPE := 1;
   #GeoAddr.IOSYSTEM := #IO_System_CP;
END_REGION

REGION Network 6: Get Hardware ID from IO System Number
   #RETVAL_GEO := GEO2LOG(GEOADDR := #GeoAddr, LADDR => #HW_ID);
END_REGION

REGION Network 7: Rack/station configured - Mode 1 - Get Configured Nodes
   // no SCL statement known for DeviceStates: written as a call
   #RETVAL_DEVICE := DeviceStates(LADDR := #HW_ID, MODE := 1, STATE := #DR_Data);
END_REGION

REGION Network 8
   MOVE_BLK(IN := #DR_Data_Trans[0], COUNT := 258, OUT => #CONFIGURED[0]);
END_REGION

REGION Network 9: Rack/station exists - Mode - 4 - Get Present Nodes
   // no SCL statement known for DeviceStates: written as a call
   #RETVAL_DEVICE_1 := DeviceStates(LADDR := #HW_ID, MODE := 4, STATE := #DR_Data);
END_REGION

REGION Network 10
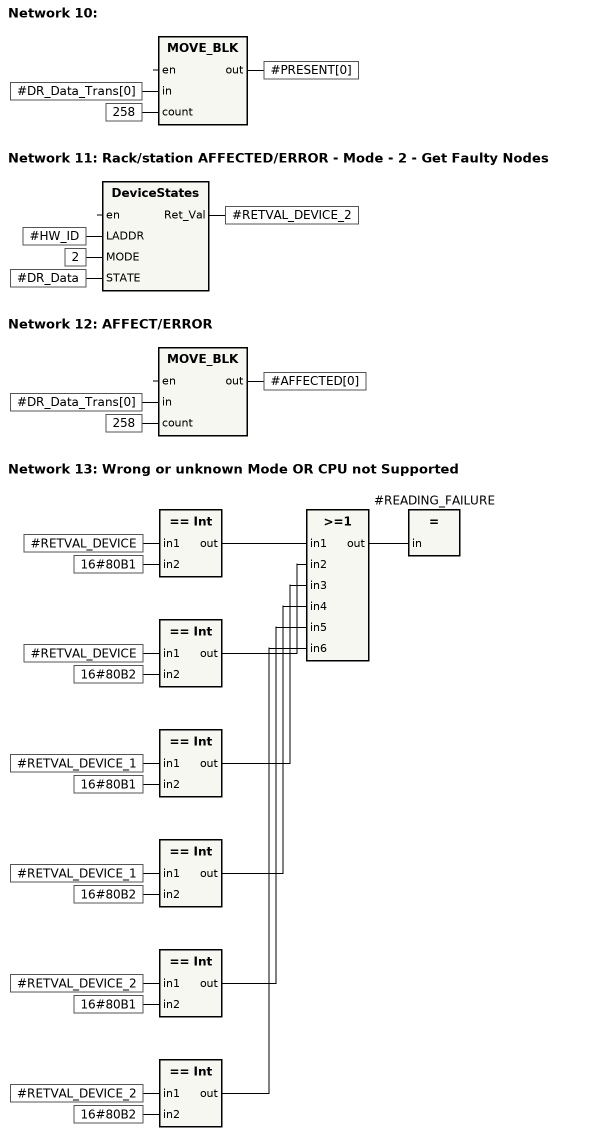
   MOVE_BLK(IN := #DR_Data_Trans[0], COUNT := 258, OUT => #PRESENT[0]);
END_REGION

REGION Network 11: Rack/station AFFECTED/ERROR - Mode - 2 - Get Faulty Nodes
   // no SCL statement known for DeviceStates: written as a call
   #RETVAL_DEVICE_2 := DeviceStates(LADDR := #HW_ID, MODE := 2, STATE := #DR_Data);
END_REGION

REGION Network 12: AFFECT/ERROR
   MOVE_BLK(IN := #DR_Data_Trans[0], COUNT := 258, OUT => #AFFECTED[0]);
END_REGION

REGION Network 13: Wrong or unknown Mode OR CPU not Supported
   // Check for Read error
   #READING_FAILURE := (#RETVAL_DEVICE = 16#80B1) OR (#RETVAL_DEVICE = 16#80B2) OR (#RETVAL_DEVICE_1 = 16#80B1) OR (#RETVAL_DEVICE_1 = 16#80B2) OR (#RETVAL_DEVICE_2 = 16#80B1) OR (#RETVAL_DEVICE_2 = 16#80B2);
END_REGION

REGION Network 14: Wrong or non permited index
   // Check for Read error
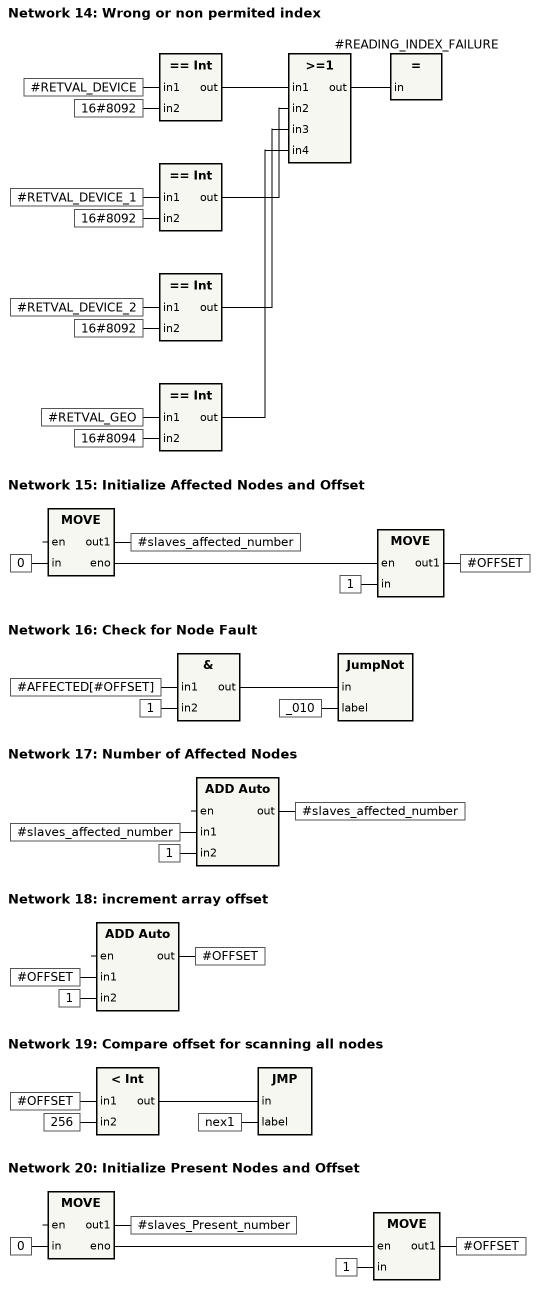
   #READING_INDEX_FAILURE := (#RETVAL_DEVICE = 16#8092) OR (#RETVAL_DEVICE_1 = 16#8092) OR (#RETVAL_DEVICE_2 = 16#8092) OR (#RETVAL_GEO = 16#8094);
END_REGION

REGION Network 15: Initialize Affected Nodes and Offset
   #slaves_affected_number := 0;
   #OFFSET := 1;
END_REGION

REGION Network 16: Check for Node Fault
   // no SCL statement known for JumpNot: written as a call
   nex1:
   JumpNot(in := #AFFECTED[#OFFSET] AND 1, label := _010);
END_REGION

REGION Network 17: Number of Affected Nodes
   #slaves_affected_number := #slaves_affected_number + 1;
END_REGION

REGION Network 18: increment array offset
   _010:
   #OFFSET := #OFFSET + 1;
END_REGION

REGION Network 19: Compare offset for scanning all nodes
   IF #OFFSET < 256 THEN GOTO nex1; END_IF;
END_REGION

REGION Network 20: Initialize Present Nodes and Offset
   #slaves_Present_number := 0;
   #OFFSET := 1;
END_REGION

REGION Network 21: Check for Node Present
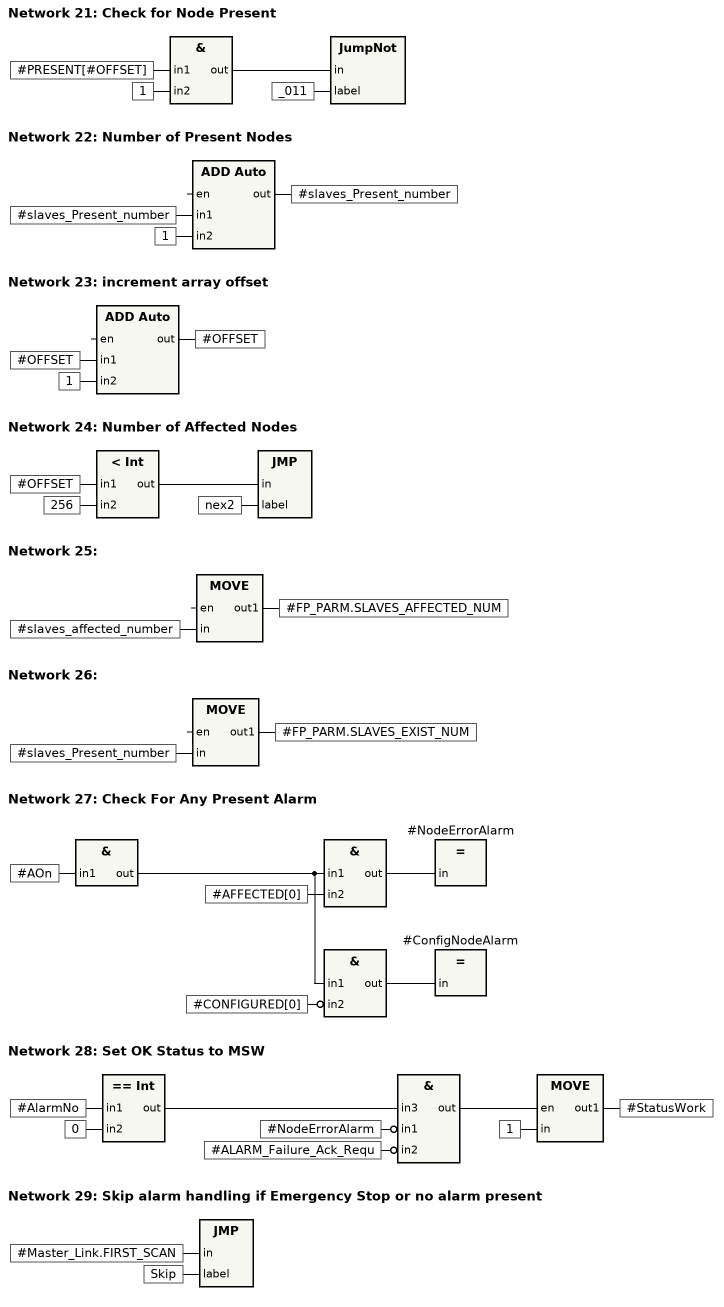
   // no SCL statement known for JumpNot: written as a call
   nex2:
   JumpNot(in := #PRESENT[#OFFSET] AND 1, label := _011);
END_REGION

REGION Network 22: Number of Present Nodes
   #slaves_Present_number := #slaves_Present_number + 1;
END_REGION

REGION Network 23: increment array offset
   _011:
   #OFFSET := #OFFSET + 1;
END_REGION

REGION Network 24: Number of Affected Nodes
   IF #OFFSET < 256 THEN GOTO nex2; END_IF;
END_REGION

REGION Network 25
   #FP_PARM.SLAVES_AFFECTED_NUM := #slaves_affected_number;
END_REGION

REGION Network 26
   #FP_PARM.SLAVES_EXIST_NUM := #slaves_Present_number;
END_REGION

REGION Network 27: Check For Any Present Alarm
   // (Bit 0 in struct = Sum of all nodes)
   #NodeErrorAlarm := #AOn AND #AFFECTED[0];
   #ConfigNodeAlarm := #AOn AND NOT #CONFIGURED[0];
END_REGION

REGION Network 28: Set OK Status to MSW
   IF (#AlarmNo = 0) AND NOT #NodeErrorAlarm AND NOT #ALARM_Failure_Ack_Requ THEN #StatusWork := 1; END_IF;
END_REGION

REGION Network 29: Skip alarm handling if Emergency Stop or no alarm present
   // Skip = Skip Alarm
   IF #Master_Link.FIRST_SCAN THEN GOTO Skip; END_IF;
END_REGION

REGION Network 30: Alarm Present
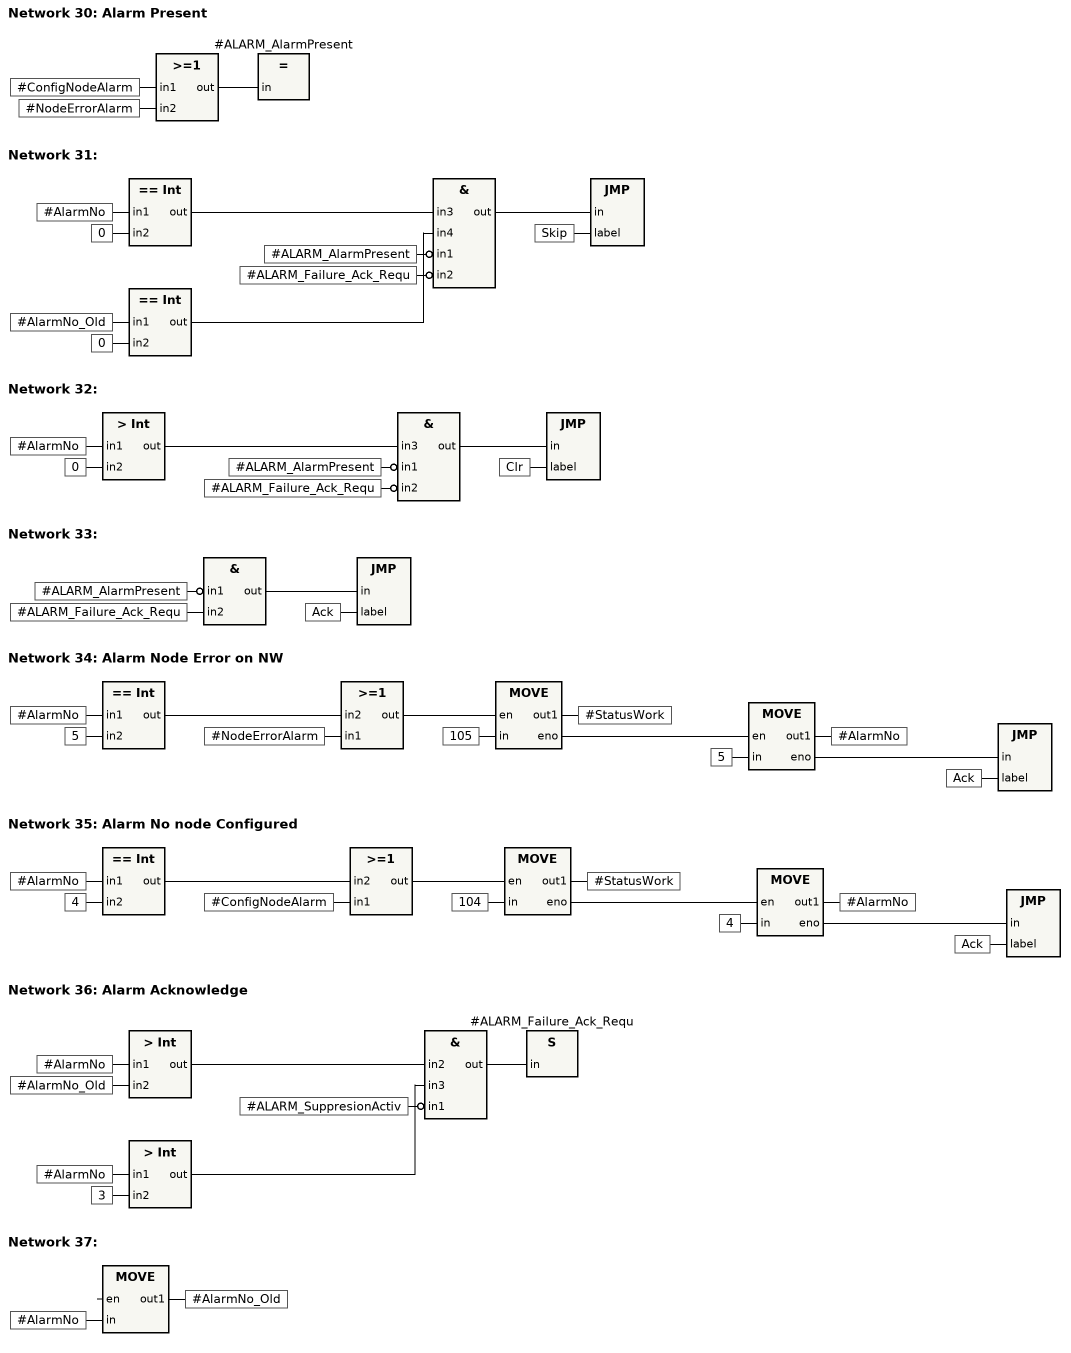
   #ALARM_AlarmPresent := #ConfigNodeAlarm OR #NodeErrorAlarm;
END_REGION

REGION Network 31
   // Skip = Skip Alarm
   IF (#AlarmNo = 0) AND (#AlarmNo_Old = 0) AND NOT #ALARM_AlarmPresent AND NOT #ALARM_Failure_Ack_Requ THEN
       GOTO Skip;
   END_IF;
END_REGION

REGION Network 32
   // Clr = Clear Alarm
   IF (#AlarmNo > 0) AND NOT #ALARM_AlarmPresent AND NOT #ALARM_Failure_Ack_Requ THEN GOTO Clr; END_IF;
END_REGION

REGION Network 33
   // Ack = Alarm Acknowledge
   IF NOT #ALARM_AlarmPresent AND #ALARM_Failure_Ack_Requ THEN GOTO Ack; END_IF;
END_REGION

REGION Network 34: Alarm Node Error on NW
   // ENO of a box is taken as its EN; it also drops when the box reports an error
   #_w1 := (#AlarmNo = 5) OR #NodeErrorAlarm;
   IF #_w1 THEN
       #StatusWork := 105;
       #AlarmNo := 5;
       GOTO Ack;
   END_IF;
END_REGION

REGION Network 35: Alarm No node Configured
   // ENO of a box is taken as its EN; it also drops when the box reports an error
   #_w1 := (#AlarmNo = 4) OR #ConfigNodeAlarm;
   IF #_w1 THEN
       #StatusWork := 104;
       #AlarmNo := 4;
       GOTO Ack;
   END_IF;
END_REGION

REGION Network 36: Alarm Acknowledge
   Ack:
   IF (#AlarmNo > #AlarmNo_Old) AND (#AlarmNo > 3) AND NOT #ALARM_SuppresionActiv THEN
       #ALARM_Failure_Ack_Requ := TRUE;
   END_IF;
END_REGION

REGION Network 37
   #AlarmNo_Old := #AlarmNo;
END_REGION

REGION Network 38
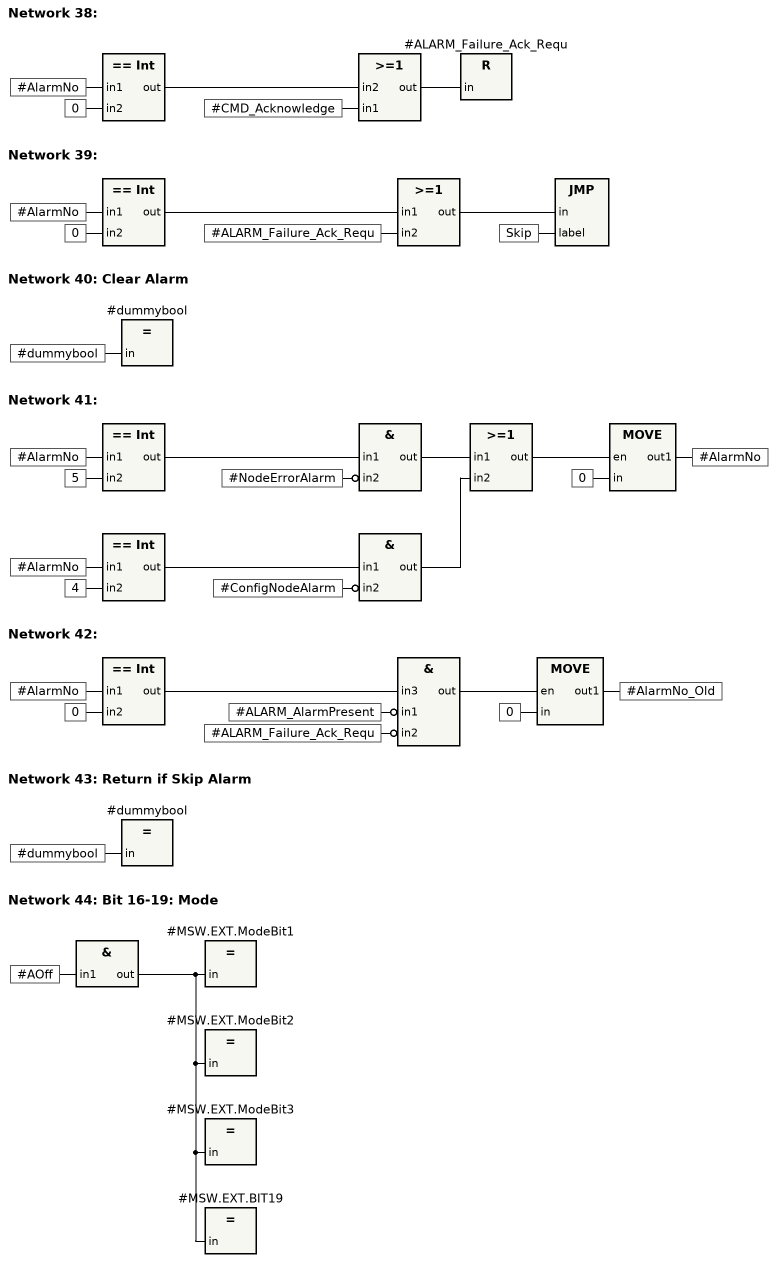
   IF (#AlarmNo = 0) OR #CMD_Acknowledge THEN #ALARM_Failure_Ack_Requ := FALSE; END_IF;
END_REGION

REGION Network 39
   // Skip = Skip Alarm
   IF (#AlarmNo = 0) OR #ALARM_Failure_Ack_Requ THEN GOTO Skip; END_IF;
END_REGION

REGION Network 40: Clear Alarm
   Clr:
   #dummybool := #dummybool;
END_REGION

REGION Network 41
   IF ((#AlarmNo = 5) AND NOT #NodeErrorAlarm) OR ((#AlarmNo = 4) AND NOT #ConfigNodeAlarm) THEN
       #AlarmNo := 0;
   END_IF;
END_REGION

REGION Network 42
   IF (#AlarmNo = 0) AND NOT #ALARM_AlarmPresent AND NOT #ALARM_Failure_Ack_Requ THEN
       #AlarmNo_Old := 0;
   END_IF;
END_REGION

REGION Network 43: Return if Skip Alarm
   Skip:
   #dummybool := #dummybool;
END_REGION

REGION Network 44: Bit 16-19: Mode
   // 0 = Auto
   // 1= Single Start
   // 2 = Manual
   // 3= Local
   // 4= Test Mode
   #MSW.EXT.ModeBit1 := #AOff;
   #MSW.EXT.ModeBit2 := #AOff;
   #MSW.EXT.ModeBit3 := #AOff;
   #MSW.EXT.BIT19 := #AOff;
END_REGION

REGION Network 45: Bit 21: Alarm Suppressed
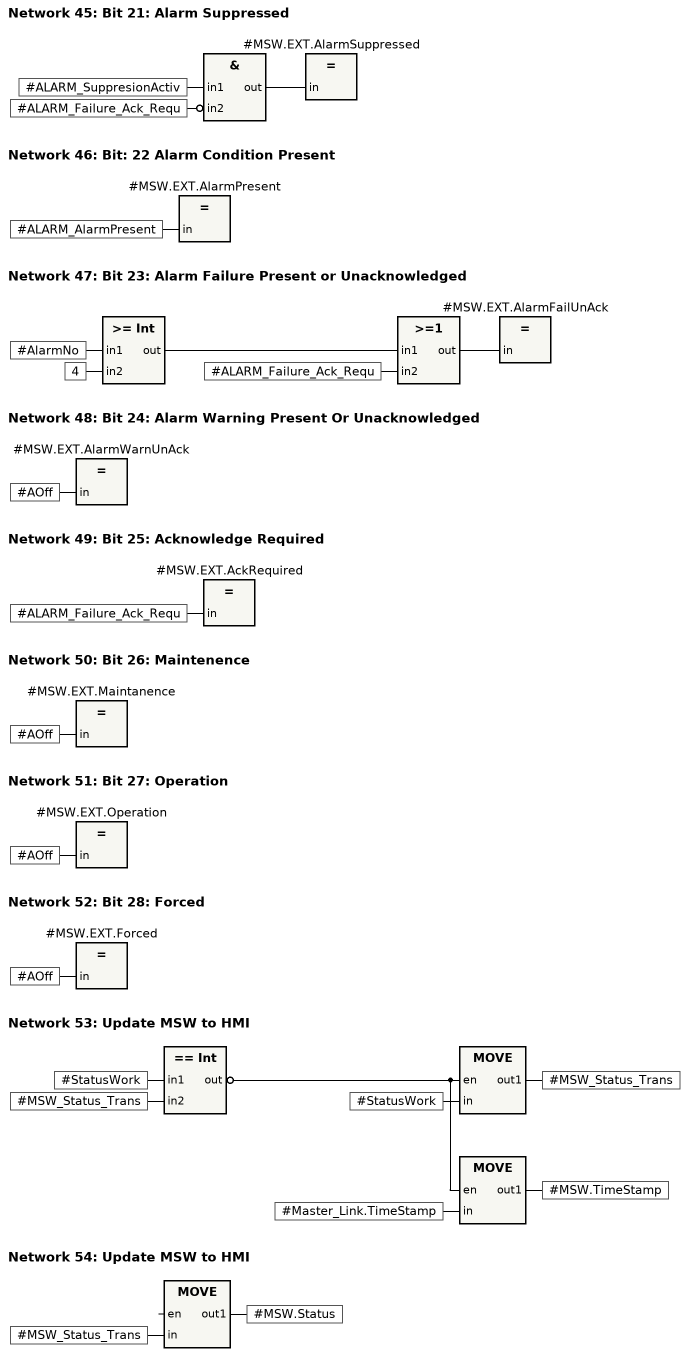
   #MSW.EXT.AlarmSuppressed := #ALARM_SuppresionActiv AND NOT #ALARM_Failure_Ack_Requ;
END_REGION

REGION Network 46: Bit: 22 Alarm Condition Present
   #MSW.EXT.AlarmPresent := #ALARM_AlarmPresent;
END_REGION

REGION Network 47: Bit 23: Alarm Failure Present or Unacknowledged
   #MSW.EXT.AlarmFailUnAck := (#AlarmNo >= 4) OR #ALARM_Failure_Ack_Requ;
END_REGION

REGION Network 48: Bit 24: Alarm Warning Present Or Unacknowledged
   #MSW.EXT.AlarmWarnUnAck := #AOff;
END_REGION

REGION Network 49: Bit 25: Acknowledge Required
   #MSW.EXT.AckRequired := #ALARM_Failure_Ack_Requ;
END_REGION

REGION Network 50: Bit 26: Maintenence
   #MSW.EXT.Maintanence := #AOff;
END_REGION

REGION Network 51: Bit 27: Operation
   #MSW.EXT.Operation := #AOff;
END_REGION

REGION Network 52: Bit 28: Forced
   #MSW.EXT.Forced := #AOff;
END_REGION

REGION Network 53: Update MSW to HMI
   #_w1 := NOT (#StatusWork = #MSW_Status_Trans);
   IF #_w1 THEN
       #MSW_Status_Trans := #StatusWork;
       #MSW.TimeStamp := #Master_Link.TimeStamp;
   END_IF;
END_REGION

REGION Network 54: Update MSW to HMI
   #MSW.Status := #MSW_Status_Trans;
END_REGION
END_FUNCTION_BLOCK

FUNCTION_BLOCK "ACESYS_PROFIBUS"   // FB224, FBD
TITLE = ACESYS V8.0 - Build 001 - Profibus Diagnostic
{ S7_Optimized_Access := 'FALSE' }
AUTHOR : FLSmidth
FAMILY : ACESYS
NAME : HWDIAG
VERSION : 8.0
   VAR_INPUT
      Master_Link : "ACESYS_MASTER_LINK";
      Enable_DPnet1_Diag : Bool;   // Enabled=1 and Disabled=0
      Int_Ext_DPnet1 : Bool;   // DPnet 1 port, External=1 and Internal=0
      DP_MasterSystemNO : Int;   // DP Master System Number
   END_VAR
   VAR_OUTPUT
      MSW : "ACESYS_HMI_STAT_32T";
   END_VAR
   VAR
      BlockInfo : Struct   // Faceplate Block Info
         Ace_Version : Int;   // Acesys Block Version Number
         Ace_BuildNo : Int;   // Acesys Block Build Number
         DB_Number : Int;   // Block Instance DB Number
      END_STRUCT;
      FP_CMD : Struct   // Faceplate Commands
         Spare_08 : Bool;   // Bit8
         Spare_09 : Bool;   // Bit9
         Spare_10 : Bool;   // Bit10
         Spare_11 : Bool;   // Bit11
         Spare_12 : Bool;   // Bit12
         Spare_13 : Bool;   // Bit13
         Spare_14 : Bool;   // Bit14
         AckAlarm : Bool;   // Alarm Acknowledge
         Spare_00 : Bool;   // Bit0
         Spare_01 : Bool;   // Bit1
         Spare_02 : Bool;   // Bit2
         Spare_03 : Bool;   // Bit3
         Spare_04 : Bool;   // Bit4
         Spare_05 : Bool;   // Bit5
         Spare_06 : Bool;   // Bit6
         Spare_07 : Bool;   // Bit7
      END_STRUCT;
      FP_PARM : Struct   // Faceplate Parameters
         NODE_IO_FAULT_NUM : Int;
         NODE_NOT_PRESENT_NUM : Int;
      END_STRUCT;
      DP1_P_Station : Array[1..128] of Bool;   // Profibus DP station Not Present, 1 = Present
      DP1_F_Station : Array[1..128] of Bool;   // Profibus DP station I/O Fault, 1 = Fault
      CONFIGURED : Array[0..129] of Bool;   // Configured Nodes, 1 = Rack/Device Configured
      DPNET1_TRIG_FC26_Spare : Bool;   // Spare
      DPNET1_BUSY_FC26_Spare : Bool;   // Spare
      DPNET1_SUM_NODE_DIAG_Spare : Int;   // Spare
      DPNET1_RET_VAL_FC26 : Int;   // Spare
      DPNET1_DATA_FIELD : Array[1..50] of Byte;   // Spare
      DR_Data : Array[0..8] of Word;
      DR_Data_Trans AT DR_Data : Array[0..143] of Bool;
      Node_IOFault_number : Int;   // Number of Nodes with IO Fault
      Loop_Counter : Int;
      OFFSET : Int;
      Nodes_NotPresent_number : Int;   // Number of non Present nodes
      StatusWork : Int;
      Node_IOFault : Bool;
      BUSY_READ_SZL_092_Spare : Bool;   // Spare
      CMD_Acknowledge : Bool;
      ALARM_AlarmPresent : Bool;
      ALARM_Failure_Ack_Requ : Bool;
      ALARM_SuppresionActiv : Bool;
      AlarmNo : Int;
      AlarmNo_Old : Int;
      Node_IO_Alarm : Bool;   // Node With IO Fault on NW
      NodeNotPresent : Bool;   // Configured Node Not Present on NW
      Node_Not_Present : Bool;
      Configured_Sum : Int;
      NodeNotPresent_SUB : Int;
      MSW_Status_Trans : Int;
   END_VAR
   VAR_TEMP
      Aon : Bool;
      Aoff : Bool;
      DummyBool : Bool;
      DATA_CONFIG_P : ANY;   // Pointer: Configured Nodes
      DB_Pointer : ANY;   // Pointer: Data Destination
      DP_MasterSystemNO_W : Word;
      TempDword : DWord;
      Addr_InstanceDB : DWord;   // Start Adress DR_Data
      RETVAL_DEVICE : Int;
      BlkMov_Status : Int;
      GeoAddr : GEOADDR;   // Structure for reading Hardware ID from PN Master No
      HW_ID : Hw_Any;
      RETVAL_GEO : Int;
      RETVAL_DEVICE_1 : Int;
      RETVAL_DEVICE_2 : Int;
   END_VAR
   VAR_TEMP   // added for the SCL form of the ladder/FBD networks
      _w1 : Bool;
   END_VAR
BEGIN

REGION Network 1
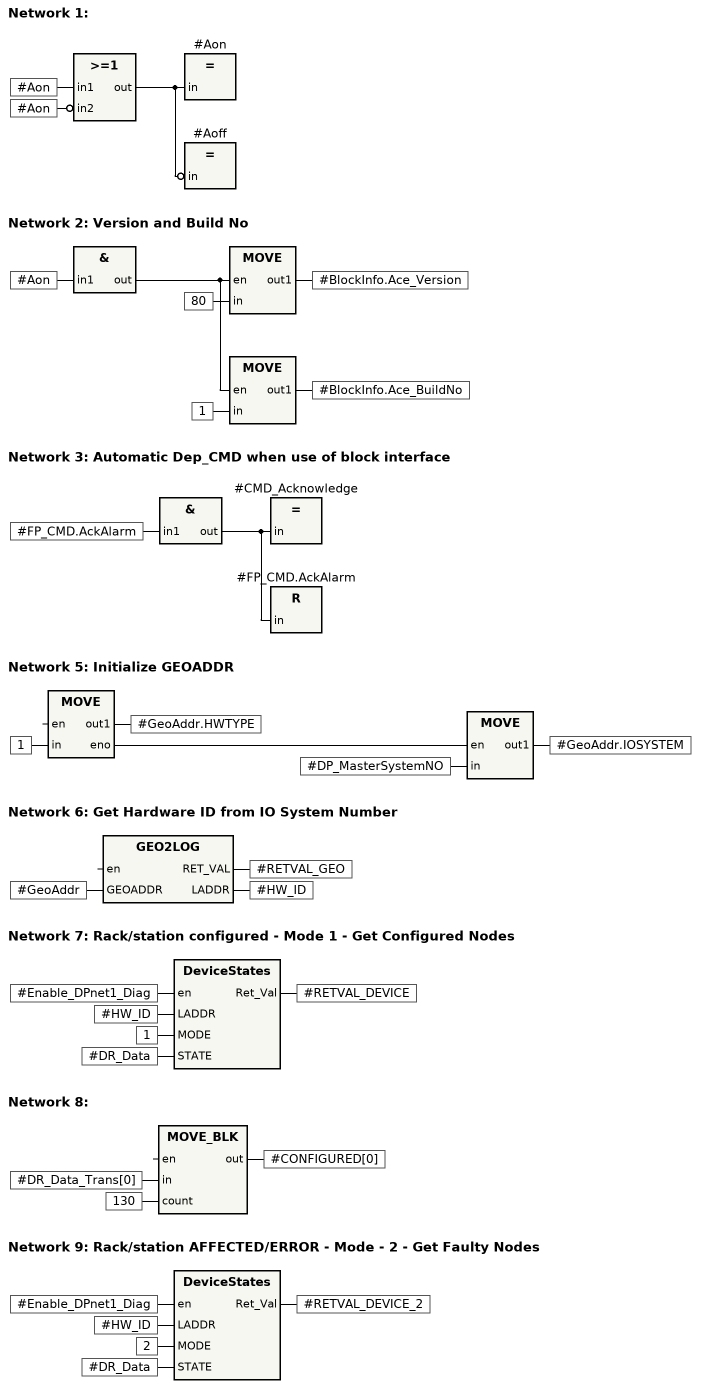
   #Aon := #Aon OR NOT #Aon;
   #Aoff := NOT #Aon;
END_REGION

REGION Network 2: Version and Build No
   IF #Aon THEN
       #BlockInfo.Ace_Version := 80;
       #BlockInfo.Ace_BuildNo := 1;
   END_IF;
END_REGION

REGION Network 3: Automatic Dep_CMD when use of block interface
   #CMD_Acknowledge := #FP_CMD.AckAlarm;
   IF #FP_CMD.AckAlarm THEN #FP_CMD.AckAlarm := FALSE; END_IF;
END_REGION

REGION Network 4 (STL): Instance DB Number to Faceplate
         L     DINO;
         T     #BlockInfo.DB_Number;
END_REGION

REGION Network 5: Initialize GEOADDR
   // ENO of a box is taken as its EN; it also drops when the box reports an error
   #GeoAddr.HWTYPE := 1;
   #GeoAddr.IOSYSTEM := #DP_MasterSystemNO;
END_REGION

REGION Network 6: Get Hardware ID from IO System Number
   #RETVAL_GEO := GEO2LOG(GEOADDR := #GeoAddr, LADDR => #HW_ID);
END_REGION

REGION Network 7: Rack/station configured - Mode 1 - Get Configured Nodes
   // no SCL statement known for DeviceStates: written as a call
   IF #Enable_DPnet1_Diag THEN
       #RETVAL_DEVICE := DeviceStates(LADDR := #HW_ID, MODE := 1, STATE := #DR_Data);
   END_IF;
END_REGION

REGION Network 8
   MOVE_BLK(IN := #DR_Data_Trans[0], COUNT := 130, OUT => #CONFIGURED[0]);
END_REGION

REGION Network 9: Rack/station AFFECTED/ERROR - Mode - 2 - Get Faulty Nodes
   // no SCL statement known for DeviceStates: written as a call
   IF #Enable_DPnet1_Diag THEN
       #RETVAL_DEVICE_2 := DeviceStates(LADDR := #HW_ID, MODE := 2, STATE := #DR_Data);
   END_IF;
END_REGION

REGION Network 10: AFFECT/ERROR
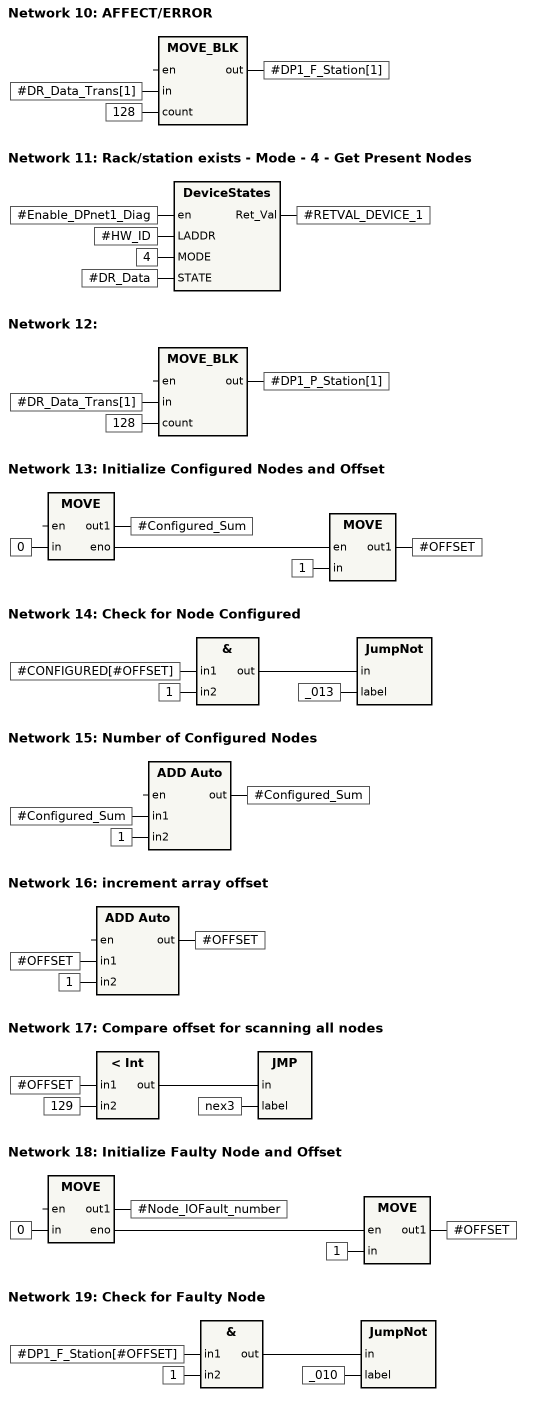
   MOVE_BLK(IN := #DR_Data_Trans[1], COUNT := 128, OUT => #DP1_F_Station[1]);
END_REGION

REGION Network 11: Rack/station exists - Mode - 4 - Get Present Nodes
   // no SCL statement known for DeviceStates: written as a call
   IF #Enable_DPnet1_Diag THEN
       #RETVAL_DEVICE_1 := DeviceStates(LADDR := #HW_ID, MODE := 4, STATE := #DR_Data);
   END_IF;
END_REGION

REGION Network 12
   MOVE_BLK(IN := #DR_Data_Trans[1], COUNT := 128, OUT => #DP1_P_Station[1]);
END_REGION

REGION Network 13: Initialize Configured Nodes and Offset
   #Configured_Sum := 0;
   #OFFSET := 1;
END_REGION

REGION Network 14: Check for Node Configured
   // no SCL statement known for JumpNot: written as a call
   nex3:
   JumpNot(in := #CONFIGURED[#OFFSET] AND 1, label := _013);
END_REGION

REGION Network 15: Number of Configured Nodes
   #Configured_Sum := #Configured_Sum + 1;
END_REGION

REGION Network 16: increment array offset
   _013:
   #OFFSET := #OFFSET + 1;
END_REGION

REGION Network 17: Compare offset for scanning all nodes
   IF #OFFSET < 129 THEN GOTO nex3; END_IF;
END_REGION

REGION Network 18: Initialize Faulty Node and Offset
   #Node_IOFault_number := 0;
   #OFFSET := 1;
END_REGION

REGION Network 19: Check for Faulty Node
   // no SCL statement known for JumpNot: written as a call
   nex1:
   JumpNot(in := #DP1_F_Station[#OFFSET] AND 1, label := _010);
END_REGION

REGION Network 20: Number of Faulty Nodes
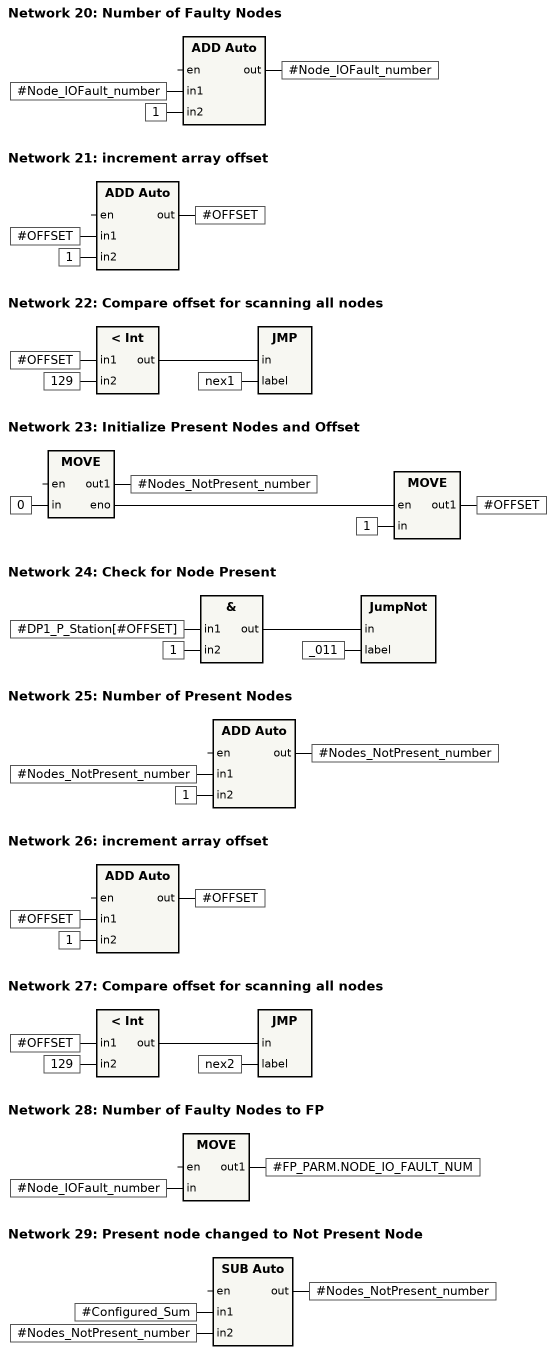
   #Node_IOFault_number := #Node_IOFault_number + 1;
END_REGION

REGION Network 21: increment array offset
   _010:
   #OFFSET := #OFFSET + 1;
END_REGION

REGION Network 22: Compare offset for scanning all nodes
   IF #OFFSET < 129 THEN GOTO nex1; END_IF;
END_REGION

REGION Network 23: Initialize Present Nodes and Offset
   #Nodes_NotPresent_number := 0;
   #OFFSET := 1;
END_REGION

REGION Network 24: Check for Node Present
   // no SCL statement known for JumpNot: written as a call
   nex2:
   JumpNot(in := #DP1_P_Station[#OFFSET] AND 1, label := _011);
END_REGION

REGION Network 25: Number of Present Nodes
   #Nodes_NotPresent_number := #Nodes_NotPresent_number + 1;
END_REGION

REGION Network 26: increment array offset
   _011:
   #OFFSET := #OFFSET + 1;
END_REGION

REGION Network 27: Compare offset for scanning all nodes
   IF #OFFSET < 129 THEN GOTO nex2; END_IF;
END_REGION

REGION Network 28: Number of Faulty Nodes to FP
   #FP_PARM.NODE_IO_FAULT_NUM := #Node_IOFault_number;
END_REGION

REGION Network 29: Present node changed to Not Present Node
   #Nodes_NotPresent_number := #Configured_Sum - #Nodes_NotPresent_number;
END_REGION

REGION Network 30: Number of not Present Nodes to FP
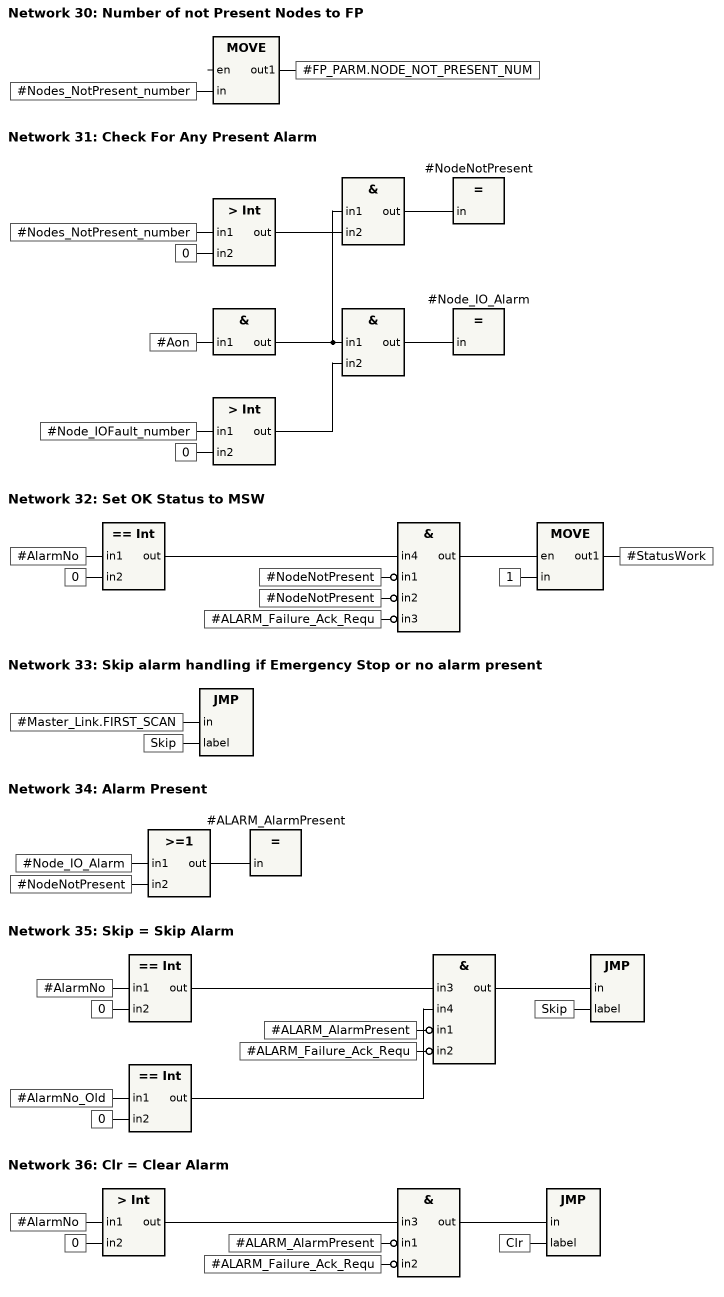
   #FP_PARM.NODE_NOT_PRESENT_NUM := #Nodes_NotPresent_number;
END_REGION

REGION Network 31: Check For Any Present Alarm
   // (Bit 0 in struct = Sum of all nodes)
   #NodeNotPresent := #Aon AND (#Nodes_NotPresent_number > 0);
   #Node_IO_Alarm := #Aon AND (#Node_IOFault_number > 0);
END_REGION

REGION Network 32: Set OK Status to MSW
   IF (#AlarmNo = 0) AND NOT #NodeNotPresent AND NOT #NodeNotPresent AND NOT #ALARM_Failure_Ack_Requ THEN
       #StatusWork := 1;
   END_IF;
END_REGION

REGION Network 33: Skip alarm handling if Emergency Stop or no alarm present
   // Skip = Skip Alarm
   IF #Master_Link.FIRST_SCAN THEN GOTO Skip; END_IF;
END_REGION

REGION Network 34: Alarm Present
   #ALARM_AlarmPresent := #Node_IO_Alarm OR #NodeNotPresent;
END_REGION

REGION Network 35: Skip = Skip Alarm
   IF (#AlarmNo = 0) AND (#AlarmNo_Old = 0) AND NOT #ALARM_AlarmPresent AND NOT #ALARM_Failure_Ack_Requ THEN
       GOTO Skip;
   END_IF;
END_REGION

REGION Network 36: Clr = Clear Alarm
   IF (#AlarmNo > 0) AND NOT #ALARM_AlarmPresent AND NOT #ALARM_Failure_Ack_Requ THEN GOTO Clr; END_IF;
END_REGION

REGION Network 37: Ack = Alarm Acknowledge
